# B&R Automation Studio project AAU12Segmenter (part 6)

#### rotationProgram.st
```iecst
ACTION rotationTask:
	positionContainerRotation[0].initXPos := 0.180;
	positionContainerRotation[0].initYPos := 0.060;
	positionContainerRotation[1].initXPos := 0.060;
	positionContainerRotation[1].initYPos := 0.060;
	positionContainerRotation[2].initXPos := 0.060;
	positionContainerRotation[2].initYPos := 0.180;
	positionContainerRotation[3].initXPos := 0.180;
	positionContainerRotation[3].initYPos := 0.180;

	positionContainerRotation[4].initXPos := 0.120;
	positionContainerRotation[4].initYPos := 0.360;
	positionContainerRotation[5].initXPos := 0.360;
	positionContainerRotation[5].initYPos := 0.360;
	positionContainerRotation[6].initXPos := 0.600;
	positionContainerRotation[6].initYPos := 0.360;
	positionContainerRotation[7].initXPos := 0.360;
	positionContainerRotation[7].initYPos := 0.600;

	gWorkStations[0].par.xLocation										:= 0.180;
	gWorkStations[0].par.yLocation										:= 0.060;
	gWorkStations[0].par.nextStationSelector							:= '1';
	gWorkStations[0].par.processTime									:= 0;
	gWorkStations[0].par.pathRouting									:= 1;
	gWorkStations[0].par.landBeforeProcess								:= FALSE;
	gWorkStations[0].par.ArcMovement									:= FALSE;

	gWorkStations[1].par.xLocation										:= 0.060;
	gWorkStations[1].par.yLocation										:= 0.180;
	gWorkStations[1].par.nextStationSelector							:= '0';
	gWorkStations[1].par.processTime									:= 2;
	gWorkStations[1].par.pathRouting									:= 1;
	gWorkStations[1].par.landBeforeProcess								:= TRUE;
	gWorkStations[1].par.ArcMovement									:= FALSE;

	CASE em.substate OF
		14000:
			em.description := 'Move shuttle to pre pos';
			tempShuttleCounter := 0;
			MC_BR_MoveInPlaneAsync_Acp6D_0.Parameters.Acceleration := gAcp6DCtrl.Par.Acceleration;
			MC_BR_MoveInPlaneAsync_Acp6D_0.Parameters.Velocity := gAcp6DCtrl.Par.Velocity;
			FOR i := 0 TO UINT_TO_USINT(localCurrentNumShuttles-1) DO
				MC_BR_MoveInPlaneAsync_Acp6D_0.Parameters.AsyncPar[i].Shuttle := ADR(gAcp6DCtrl.Status.ShuttleInfo[i].shuttleRef);
				MC_BR_MoveInPlaneAsync_Acp6D_0.Parameters.AsyncPar[i].X := positionContainerRotation[i].initXPos;
				MC_BR_MoveInPlaneAsync_Acp6D_0.Parameters.AsyncPar[i].Y := positionContainerRotation[i].initYPos;
			END_FOR
			MC_BR_MoveInPlaneAsync_Acp6D_0.Execute := TRUE;
			IF MC_BR_MoveInPlaneAsync_Acp6D_0.Done THEN
				MC_BR_MoveInPlaneAsync_Acp6D_0.Execute := FALSE;
				tempShuttleCounter := 4;
				em.substate := 14005;
			END_IF

		14005:
			em.description := 'Start rotation of shuttle 5-10';
			IF tempShuttleCounter > localCurrentNumShuttles-1 THEN
				tempShuttleCounter := 0;
				em.substate := 14010;
			ELSE
				MC_BR_RotaryMotionSpin_Acp6D_0.Shuttle := ADR(gAcp6DCtrl.Status.ShuttleInfo[tempShuttleCounter].shuttleRef);
				MC_BR_RotaryMotionSpin_Acp6D_0.Parameters.Acceleration := gAcp6DCtrl.Par.rotationAcceleration;
				MC_BR_RotaryMotionSpin_Acp6D_0.Parameters.Velocity := gAcp6DCtrl.Par.rotationVelocity;
				MC_BR_RotaryMotionSpin_Acp6D_0.Parameters.Duration := 1000;
				MC_BR_RotaryMotionSpin_Acp6D_0.Execute := TRUE;
				IF MC_BR_RotaryMotionSpin_Acp6D_0.Acknowledge THEN
					MC_BR_RotaryMotionSpin_Acp6D_0.Execute := FALSE;
					em.substate := 14006;
				END_IF
			END_IF

		14006:
			em.description := 'Dummy scan';
			TON_0.PT := t#2s;
			TON_0.IN := TRUE;
			IF TON_0.Q THEN
				TON_0.IN := FALSE;
				tempShuttleCounter := tempShuttleCounter + 1;
				em.substate := 14005;
			END_IF

		14010:
			em.description := 'Move shuttle 2 towards workstation 0';
			MC_BR_MoveInPlane_Acp6D_0.Parameters.Acceleration := gAcp6DCtrl.Par.Acceleration;
			MC_BR_MoveInPlane_Acp6D_0.Parameters.Velocity := gAcp6DCtrl.Par.Velocity;
			MC_BR_MoveInPlane_Acp6D_0.Shuttle := ADR(gAcp6DCtrl.Status.ShuttleInfo[1].shuttleRef);;
			MC_BR_MoveInPlane_Acp6D_0.Parameters.Position.X := gWorkStations[0].par.xLocation;;
			MC_BR_MoveInPlane_Acp6D_0.Parameters.Position.Y := gWorkStations[0].par.yLocation;
			MC_BR_MoveInPlane_Acp6D_0.Parameters.Path := 0; //direct
			MC_BR_MoveInPlane_Acp6D_0.Parameters.Mode := 0;
			MC_BR_MoveInPlane_Acp6D_0.Execute := TRUE;
			IF MC_BR_MoveInPlane_Acp6D_0.Acknowledge THEN
				MC_BR_MoveInPlane_Acp6D_0.Execute := FALSE;
				em.substate := 14020;
			END_IF

		14020:
			em.description := 'Move shuttle 3 towards workstation 0';
			MC_BR_MoveInPlane_Acp6D_0.Parameters.Acceleration := gAcp6DCtrl.Par.Acceleration;
			MC_BR_MoveInPlane_Acp6D_0.Parameters.Velocity := gAcp6DCtrl.Par.Velocity;
			MC_BR_MoveInPlane_Acp6D_0.Shuttle := ADR(gAcp6DCtrl.Status.ShuttleInfo[2].shuttleRef);;
			MC_BR_MoveInPlane_Acp6D_0.Parameters.Position.X := gWorkStations[0].par.xLocation;;
			MC_BR_MoveInPlane_Acp6D_0.Parameters.Position.Y := gWorkStations[0].par.yLocation;
			MC_BR_MoveInPlane_Acp6D_0.Parameters.Path := 2; //Y then X
			MC_BR_MoveInPlane_Acp6D_0.Parameters.Mode := 0;
			MC_BR_MoveInPlane_Acp6D_0.Execute := TRUE;
			IF MC_BR_MoveInPlane_Acp6D_0.Acknowledge THEN
				MC_BR_MoveInPlane_Acp6D_0.Execute := FALSE;
				em.substate := 14030;
			END_IF

		14030:
			em.description := 'Move shuttle 4 towards workstation 1';
			MC_BR_MoveInPlane_Acp6D_0.Parameters.Acceleration := gAcp6DCtrl.Par.Acceleration;
			MC_BR_MoveInPlane_Acp6D_0.Parameters.Velocity := gAcp6DCtrl.Par.Velocity;
			MC_BR_MoveInPlane_Acp6D_0.Shuttle := ADR(gAcp6DCtrl.Status.ShuttleInfo[3].shuttleRef);;
			MC_BR_MoveInPlane_Acp6D_0.Parameters.Position.X := 0.060;
			MC_BR_MoveInPlane_Acp6D_0.Parameters.Position.Y := 0.180;
			MC_BR_MoveInPlane_Acp6D_0.Parameters.Path := 0; //direct
			MC_BR_MoveInPlane_Acp6D_0.Parameters.Mode := 0;
			MC_BR_MoveInPlane_Acp6D_0.Execute := TRUE;
			IF MC_BR_MoveInPlane_Acp6D_0.Acknowledge THEN
				MC_BR_MoveInPlane_Acp6D_0.Execute := FALSE;
				em.substate := 14040;
			END_IF

		14040:
			em.description := 'Move shuttle 4 towards workstation 1';
			MC_BR_MoveInPlane_Acp6D_0.Parameters.Acceleration := gAcp6DCtrl.Par.Acceleration;
			MC_BR_MoveInPlane_Acp6D_0.Parameters.Velocity := gAcp6DCtrl.Par.Velocity;
			MC_BR_MoveInPlane_Acp6D_0.Shuttle := ADR(gAcp6DCtrl.Status.ShuttleInfo[3].shuttleRef);;
			MC_BR_MoveInPlane_Acp6D_0.Parameters.Position.X := gWorkStations[0].par.xLocation;
			MC_BR_MoveInPlane_Acp6D_0.Parameters.Position.Y := gWorkStations[0].par.yLocation;
			MC_BR_MoveInPlane_Acp6D_0.Parameters.Path := 2; //direct
			MC_BR_MoveInPlane_Acp6D_0.Parameters.Mode := 0;
			MC_BR_MoveInPlane_Acp6D_0.Execute := TRUE;
			IF MC_BR_MoveInPlane_Acp6D_0.Acknowledge THEN
				MC_BR_MoveInPlane_Acp6D_0.Execute := FALSE;
				em.substate := 14050;
			END_IF

		14050:
			IF em.status.parent.state <> STATE_EXECUTE THEN
				em.substate := 14060;
			END_IF

		14060:
			MC_BR_AsmStop_Acp6D_0.Execute := TRUE;
			IF MC_BR_AsmStop_Acp6D_0.Done THEN
				MC_BR_AsmStop_Acp6D_0.Execute := FALSE;
				em.substate := 14070;
			END_IF

		14070:
			// Wait for shuttles to settle after rotation
			TON_0.PT := t#2s;
			TON_0.IN := TRUE;
			IF TON_0.Q THEN
				TON_0.IN := FALSE;
				tempShuttleCounter := 4;
				em.substate := 14080;
			END_IF

		14080:
			em.description := 'Start rotation of shuttle 5-10';
			IF tempShuttleCounter > localCurrentNumShuttles-1 THEN
				tempShuttleCounter := 0;
				em.substate := 14100;
			ELSIF gAcp6DCtrl.Status.ShuttleInfo[tempShuttleCounter].State = mcACP6D_SH_STATE_IDLING THEN
				MC_BR_RotaryMotion_Acp6D_0.Shuttle := ADR(gAcp6DCtrl.Status.ShuttleInfo[tempShuttleCounter].shuttleRef);
				MC_BR_RotaryMotion_Acp6D_0.Parameters.Acceleration := gAcp6DCtrl.Par.rotationAcceleration;
				MC_BR_RotaryMotion_Acp6D_0.Parameters.Velocity := gAcp6DCtrl.Par.rotationVelocity;
				MC_BR_RotaryMotion_Acp6D_0.Parameters.Mode := mcACP6D_ROTATE_CLOCKWISE;
				MC_BR_RotaryMotion_Acp6D_0.Parameters.Angle := 0;
				MC_BR_RotaryMotion_Acp6D_0.Execute := TRUE;
				IF MC_BR_RotaryMotion_Acp6D_0.Done THEN
					MC_BR_RotaryMotion_Acp6D_0.Execute := FALSE;
					em.substate := 14090;
				END_IF
			END_IF

		14090:
			em.description := 'Dummyscan';
			tempShuttleCounter := tempShuttleCounter + 1;
			em.substate := 14080;

		14100:
			em.description := 'check all shuttles that is rotating to pos zero is done';
			FOR i := 4 TO NUM_SHUTTLES DO
				IF gAcp6DCtrl.Status.ShuttleInfo[i].State = mcACP6D_SH_STATE_IDLING THEN
				ELSE
					EXIT;
				END_IF
			END_FOR
			IF i > NUM_SHUTTLES THEN
				em.substate := 14110;
			END_IF

		14110:
			em.cmd.sc := TRUE;

	END_CASE

END_ACTION

ACTION rotationStation:
	CASE cm.state OF
		// Display station at image
		//'<foreignObject x="20" y="20" width="300" height="300"><img src="Media/statusGreen.png" height="300" width="300"/>'
		//brsstrcat(ADR(showWorkStations),ADR('<foreingObject x="'));
		//brdkStrCat(ADR(showWorkStations), ADR(testDraw));
		//brdkStrCat(ADR(showWorkStations),'<foreingObject x="');

		0:
			//Check what shuttle is on top of workstation
			FOR k := 0 TO NUM_SHUTTLES DO
				IF((gAcp6DCtrl.Status.ShuttleInfo[k].Position.X > pWorkStations.par.xLocation - MARGIN AND gAcp6DCtrl.Status.ShuttleInfo[k].Position.X < pWorkStations.par.xLocation + MARGIN) AND
					gAcp6DCtrl.Status.ShuttleInfo[k].Position.Y > pWorkStations.par.yLocation - MARGIN AND gAcp6DCtrl.Status.ShuttleInfo[k].Position.Y < pWorkStations.par.yLocation + MARGIN) THEN
					IF gAcp6DCtrl.Status.ShuttleInfo[k].State = mcACP6D_SH_STATE_IDLING THEN
						pWorkStations.par.tempShuttleID := k;
						cm.state := 10;
					END_IF
				END_IF
			END_FOR

		10:
			//Move first workstation
			pWorkStations.MC_BR_MoveInPlane_Acp6D_0.Shuttle := ADR(gAcp6DCtrl.Status.ShuttleInfo[pWorkStations.par.tempShuttleID].shuttleRef);
			pWorkStations.MC_BR_MoveInPlane_Acp6D_0.Parameters.Velocity := gAcp6DCtrl.Par.Velocity;
			pWorkStations.MC_BR_MoveInPlane_Acp6D_0.Parameters.Acceleration := gAcp6DCtrl.Par.Acceleration;
			pWorkStations.MC_BR_MoveInPlane_Acp6D_0.Parameters.Position.X := 0.360;
			pWorkStations.MC_BR_MoveInPlane_Acp6D_0.Parameters.Position.Y := 0.120;
			pWorkStations.MC_BR_MoveInPlane_Acp6D_0.Parameters.Mode := 0; //Absolute
			pWorkStations.MC_BR_MoveInPlane_Acp6D_0.Parameters.Path := 1; //0 Diagonal, 1 First X then Y, 2 First Y then X
			pWorkStations.MC_BR_MoveInPlane_Acp6D_0.Execute := TRUE;
			IF pWorkStations.MC_BR_MoveInPlane_Acp6D_0.Done THEN
				pWorkStations.MC_BR_MoveInPlane_Acp6D_0.Execute := FALSE;
				cm.state := 20;
			END_IF

		20:
			//Rotate 90 degress
			em.cmd.sc := FALSE;
			pWorkStations.MC_BR_RotaryMotion_Acp6D_0.Shuttle := ADR(gAcp6DCtrl.Status.ShuttleInfo[pWorkStations.par.tempShuttleID].shuttleRef);
			pWorkStations.MC_BR_RotaryMotion_Acp6D_0.Parameters.Acceleration := gAcp6DCtrl.Par.rotationAcceleration;
			pWorkStations.MC_BR_RotaryMotion_Acp6D_0.Parameters.Velocity := gAcp6DCtrl.Par.rotationVelocity;
			pWorkStations.MC_BR_RotaryMotion_Acp6D_0.Parameters.Angle := 1.57079633; //90 degress
			pWorkStations.MC_BR_RotaryMotion_Acp6D_0.Parameters.Mode := 0;
			pWorkStations.MC_BR_RotaryMotion_Acp6D_0.Execute := TRUE;
			IF pWorkStations.MC_BR_RotaryMotion_Acp6D_0.Done THEN
				pWorkStations.MC_BR_RotaryMotion_Acp6D_0.Execute := FALSE;
				cm.state := 30;
			END_IF

		30:
			//Move
			pWorkStations.MC_BR_MoveInPlane_Acp6D_0.Shuttle := ADR(gAcp6DCtrl.Status.ShuttleInfo[pWorkStations.par.tempShuttleID].shuttleRef);
			pWorkStations.MC_BR_MoveInPlane_Acp6D_0.Parameters.Velocity := gAcp6DCtrl.Par.Velocity;
			pWorkStations.MC_BR_MoveInPlane_Acp6D_0.Parameters.Acceleration := gAcp6DCtrl.Par.Acceleration;
			pWorkStations.MC_BR_MoveInPlane_Acp6D_0.Parameters.Position.X := 0.420;
			pWorkStations.MC_BR_MoveInPlane_Acp6D_0.Parameters.Position.Y := 0.120;
			pWorkStations.MC_BR_MoveInPlane_Acp6D_0.Parameters.Mode := 0; //Absolute
			pWorkStations.MC_BR_MoveInPlane_Acp6D_0.Parameters.Path := 1; //0 Diagonal, 1 First X then Y, 2 First Y then X
			pWorkStations.MC_BR_MoveInPlane_Acp6D_0.Execute := TRUE;
			IF pWorkStations.MC_BR_MoveInPlane_Acp6D_0.Acknowledge THEN
				pWorkStations.MC_BR_MoveInPlane_Acp6D_0.Execute := FALSE;
				cm.state := 40;
			END_IF

		40:
			pWorkStations.TON_0.IN := TRUE;
			pWorkStations.TON_0.PT := t#1s;
			IF pWorkStations.TON_0.Q THEN
				pWorkStations.TON_0.IN := FALSE;
				cm.state := 50;
			END_IF

		50:
			//Move
			pWorkStations.MC_BR_MoveInPlane_Acp6D_0.Shuttle := ADR(gAcp6DCtrl.Status.ShuttleInfo[pWorkStations.par.tempShuttleID].shuttleRef);
			pWorkStations.MC_BR_MoveInPlane_Acp6D_0.Parameters.Velocity := gAcp6DCtrl.Par.Velocity;
			pWorkStations.MC_BR_MoveInPlane_Acp6D_0.Parameters.Acceleration := gAcp6DCtrl.Par.Acceleration;
			pWorkStations.MC_BR_MoveInPlane_Acp6D_0.Parameters.Position.X := 0.360;
			pWorkStations.MC_BR_MoveInPlane_Acp6D_0.Parameters.Position.Y := 0.120;
			pWorkStations.MC_BR_MoveInPlane_Acp6D_0.Parameters.Mode := 0; //Absolute
			pWorkStations.MC_BR_MoveInPlane_Acp6D_0.Parameters.Path := 1; //0 Diagonal, 1 First X then Y, 2 First Y then X
			pWorkStations.MC_BR_MoveInPlane_Acp6D_0.Execute := TRUE;
			IF pWorkStations.MC_BR_MoveInPlane_Acp6D_0.Acknowledge THEN
				pWorkStations.MC_BR_MoveInPlane_Acp6D_0.Execute := FALSE;
				cm.state := 60;
			END_IF

		60:
			//Rotate 90 degress
			em.cmd.sc := FALSE;
			pWorkStations.MC_BR_RotaryMotion_Acp6D_0.Shuttle := ADR(gAcp6DCtrl.Status.ShuttleInfo[pWorkStations.par.tempShuttleID].shuttleRef);
			pWorkStations.MC_BR_RotaryMotion_Acp6D_0.Parameters.Acceleration := gAcp6DCtrl.Par.rotationAcceleration;
			pWorkStations.MC_BR_RotaryMotion_Acp6D_0.Parameters.Velocity := gAcp6DCtrl.Par.rotationVelocity;
			pWorkStations.MC_BR_RotaryMotion_Acp6D_0.Parameters.Angle := 3.14159265; //180 degress
			pWorkStations.MC_BR_RotaryMotion_Acp6D_0.Parameters.Mode := 0;
			pWorkStations.MC_BR_RotaryMotion_Acp6D_0.Execute := TRUE;
			IF pWorkStations.MC_BR_RotaryMotion_Acp6D_0.Done THEN
				pWorkStations.MC_BR_RotaryMotion_Acp6D_0.Execute := FALSE;
				cm.state := 70;
			END_IF

		70:
			//Move
			pWorkStations.MC_BR_MoveInPlane_Acp6D_0.Shuttle := ADR(gAcp6DCtrl.Status.ShuttleInfo[pWorkStations.par.tempShuttleID].shuttleRef);
			pWorkStations.MC_BR_MoveInPlane_Acp6D_0.Parameters.Velocity := gAcp6DCtrl.Par.Velocity;
			pWorkStations.MC_BR_MoveInPlane_Acp6D_0.Parameters.Acceleration := gAcp6DCtrl.Par.Acceleration;
			pWorkStations.MC_BR_MoveInPlane_Acp6D_0.Parameters.Position.X := 0.420;
			pWorkStations.MC_BR_MoveInPlane_Acp6D_0.Parameters.Position.Y := 0.120;
			pWorkStations.MC_BR_MoveInPlane_Acp6D_0.Parameters.Mode := 0; //Absolute
			pWorkStations.MC_BR_MoveInPlane_Acp6D_0.Parameters.Path := 1; //0 Diagonal, 1 First X then Y, 2 First Y then X
			pWorkStations.MC_BR_MoveInPlane_Acp6D_0.Execute := TRUE;
			IF pWorkStations.MC_BR_MoveInPlane_Acp6D_0.Acknowledge THEN
				pWorkStations.MC_BR_MoveInPlane_Acp6D_0.Execute := FALSE;
				cm.state := 80;
			END_IF

		80:
			pWorkStations.TON_0.IN := TRUE;
			pWorkStations.TON_0.PT := t#1s;
			IF pWorkStations.TON_0.Q THEN
				pWorkStations.TON_0.IN := FALSE;
				cm.state := 90;
			END_IF

		90:
			//Move
			pWorkStations.MC_BR_MoveInPlane_Acp6D_0.Shuttle := ADR(gAcp6DCtrl.Status.ShuttleInfo[pWorkStations.par.tempShuttleID].shuttleRef);
			pWorkStations.MC_BR_MoveInPlane_Acp6D_0.Parameters.Velocity := gAcp6DCtrl.Par.Velocity;
			pWorkStations.MC_BR_MoveInPlane_Acp6D_0.Parameters.Acceleration := gAcp6DCtrl.Par.Acceleration;
			pWorkStations.MC_BR_MoveInPlane_Acp6D_0.Parameters.Position.X := 0.360;
			pWorkStations.MC_BR_MoveInPlane_Acp6D_0.Parameters.Position.Y := 0.120;
			pWorkStations.MC_BR_MoveInPlane_Acp6D_0.Parameters.Mode := 0; //Absolute
			pWorkStations.MC_BR_MoveInPlane_Acp6D_0.Parameters.Path := 1; //0 Diagonal, 1 First X then Y, 2 First Y then X
			pWorkStations.MC_BR_MoveInPlane_Acp6D_0.Execute := TRUE;
			IF pWorkStations.MC_BR_MoveInPlane_Acp6D_0.Acknowledge THEN
				pWorkStations.MC_BR_MoveInPlane_Acp6D_0.Execute := FALSE;
				cm.state := 100;
			END_IF

		100:
			//Rotate 90 degress
			em.cmd.sc := FALSE;
			pWorkStations.MC_BR_RotaryMotion_Acp6D_0.Shuttle := ADR(gAcp6DCtrl.Status.ShuttleInfo[pWorkStations.par.tempShuttleID].shuttleRef);
			pWorkStations.MC_BR_RotaryMotion_Acp6D_0.Parameters.Acceleration := gAcp6DCtrl.Par.rotationAcceleration;
			pWorkStations.MC_BR_RotaryMotion_Acp6D_0.Parameters.Velocity := gAcp6DCtrl.Par.rotationVelocity;
			pWorkStations.MC_BR_RotaryMotion_Acp6D_0.Parameters.Angle := 4.71238898; //270 degress
			pWorkStations.MC_BR_RotaryMotion_Acp6D_0.Parameters.Mode := 0;
			pWorkStations.MC_BR_RotaryMotion_Acp6D_0.Execute := TRUE;
			IF pWorkStations.MC_BR_RotaryMotion_Acp6D_0.Done THEN
				pWorkStations.MC_BR_RotaryMotion_Acp6D_0.Execute := FALSE;
				cm.state := 110;
			END_IF

		110:
			//Move
			pWorkStations.MC_BR_MoveInPlane_Acp6D_0.Shuttle := ADR(gAcp6DCtrl.Status.ShuttleInfo[pWorkStations.par.tempShuttleID].shuttleRef);
			pWorkStations.MC_BR_MoveInPlane_Acp6D_0.Parameters.Velocity := gAcp6DCtrl.Par.Velocity;
			pWorkStations.MC_BR_MoveInPlane_Acp6D_0.Parameters.Acceleration := gAcp6DCtrl.Par.Acceleration;
			pWorkStations.MC_BR_MoveInPlane_Acp6D_0.Parameters.Position.X := 0.420;
			pWorkStations.MC_BR_MoveInPlane_Acp6D_0.Parameters.Position.Y := 0.120;
			pWorkStations.MC_BR_MoveInPlane_Acp6D_0.Parameters.Mode := 0; //Absolute
			pWorkStations.MC_BR_MoveInPlane_Acp6D_0.Parameters.Path := 1; //0 Diagonal, 1 First X then Y, 2 First Y then X
			pWorkStations.MC_BR_MoveInPlane_Acp6D_0.Execute := TRUE;
			IF pWorkStations.MC_BR_MoveInPlane_Acp6D_0.Acknowledge THEN
				pWorkStations.MC_BR_MoveInPlane_Acp6D_0.Execute := FALSE;
				cm.state := 120;
			END_IF

		120:
			pWorkStations.TON_0.IN := TRUE;
			pWorkStations.TON_0.PT := t#1s;
			IF pWorkStations.TON_0.Q THEN
				pWorkStations.TON_0.IN := FALSE;
				cm.state := 130;
			END_IF

		130:
			//Move
			pWorkStations.MC_BR_MoveInPlane_Acp6D_0.Shuttle := ADR(gAcp6DCtrl.Status.ShuttleInfo[pWorkStations.par.tempShuttleID].shuttleRef);
			pWorkStations.MC_BR_MoveInPlane_Acp6D_0.Parameters.Velocity := gAcp6DCtrl.Par.Velocity;
			pWorkStations.MC_BR_MoveInPlane_Acp6D_0.Parameters.Acceleration := gAcp6DCtrl.Par.Acceleration;
			pWorkStations.MC_BR_MoveInPlane_Acp6D_0.Parameters.Position.X := 0.360;
			pWorkStations.MC_BR_MoveInPlane_Acp6D_0.Parameters.Position.Y := 0.120;
			pWorkStations.MC_BR_MoveInPlane_Acp6D_0.Parameters.Mode := 0; //Absolute
			pWorkStations.MC_BR_MoveInPlane_Acp6D_0.Parameters.Path := 1; //0 Diagonal, 1 First X then Y, 2 First Y then X
			pWorkStations.MC_BR_MoveInPlane_Acp6D_0.Execute := TRUE;
			IF pWorkStations.MC_BR_MoveInPlane_Acp6D_0.Acknowledge THEN
				pWorkStations.MC_BR_MoveInPlane_Acp6D_0.Execute := FALSE;
				cm.state := 140;
			END_IF

		140:
			//Rotate
			em.cmd.sc := FALSE;
			pWorkStations.MC_BR_RotaryMotion_Acp6D_0.Shuttle := ADR(gAcp6DCtrl.Status.ShuttleInfo[pWorkStations.par.tempShuttleID].shuttleRef);
			pWorkStations.MC_BR_RotaryMotion_Acp6D_0.Parameters.Acceleration := gAcp6DCtrl.Par.rotationAcceleration;
			pWorkStations.MC_BR_RotaryMotion_Acp6D_0.Parameters.Velocity := gAcp6DCtrl.Par.rotationVelocity; //RPM
			pWorkStations.MC_BR_RotaryMotion_Acp6D_0.Parameters.Angle := 0; //0 degress
			pWorkStations.MC_BR_RotaryMotion_Acp6D_0.Parameters.Mode := 1;
			pWorkStations.MC_BR_RotaryMotion_Acp6D_0.Execute := TRUE;
			IF pWorkStations.MC_BR_RotaryMotion_Acp6D_0.Done THEN
				pWorkStations.MC_BR_RotaryMotion_Acp6D_0.Execute := FALSE;
				cm.state := 150;
			END_IF

//		145:
//			em.cmd.sc := FALSE;
//			pWorkStations.MC_BR_RotaryMotionSpin_Acp6D_0.Shuttle := ADR(gAcp6DCtrl.Status.ShuttleInfo[pWorkStations.par.tempShuttleID].shuttleRef);
//			pWorkStations.MC_BR_RotaryMotionSpin_Acp6D_0.Parameters.Acceleration := gAcp6DCtrl.Par.Acceleration;
//			pWorkStations.MC_BR_RotaryMotionSpin_Acp6D_0.Parameters.Velocity := 200; //RPM
//			pWorkStations.MC_BR_RotaryMotionSpin_Acp6D_0.Parameters.Duration := 5;
//			pWorkStations.MC_BR_RotaryMotionSpin_Acp6D_0.Execute := TRUE;
//			IF pWorkStations.MC_BR_RotaryMotionSpin_Acp6D_0.Done THEN
//				pWorkStations.MC_BR_RotaryMotionSpin_Acp6D_0.Execute := FALSE;
//				cm.state := 150;
//			END_IF

		150:
			//Move
			pWorkStations.MC_BR_MoveInPlane_Acp6D_0.Shuttle := ADR(gAcp6DCtrl.Status.ShuttleInfo[pWorkStations.par.tempShuttleID].shuttleRef);
			pWorkStations.MC_BR_MoveInPlane_Acp6D_0.Parameters.Velocity := gAcp6DCtrl.Par.Velocity;
			pWorkStations.MC_BR_MoveInPlane_Acp6D_0.Parameters.Acceleration := gAcp6DCtrl.Par.Acceleration;
			pWorkStations.MC_BR_MoveInPlane_Acp6D_0.Parameters.Position.X := 0.060;
			pWorkStations.MC_BR_MoveInPlane_Acp6D_0.Parameters.Position.Y := 0.180;
			pWorkStations.MC_BR_MoveInPlane_Acp6D_0.Parameters.Mode := 0; //Absolute
			pWorkStations.MC_BR_MoveInPlane_Acp6D_0.Parameters.Path := 2; //0 Diagonal, 1 First X then Y, 2 First Y then X
			pWorkStations.MC_BR_MoveInPlane_Acp6D_0.Execute := TRUE;
			IF pWorkStations.MC_BR_MoveInPlane_Acp6D_0.Acknowledge THEN
				pWorkStations.MC_BR_MoveInPlane_Acp6D_0.Execute := FALSE;
				cm.state := 160;
			END_IF

		160:
			//Move
			pWorkStations.MC_BR_MoveInPlane_Acp6D_0.Shuttle := ADR(gAcp6DCtrl.Status.ShuttleInfo[pWorkStations.par.tempShuttleID].shuttleRef);
			pWorkStations.MC_BR_MoveInPlane_Acp6D_0.Parameters.Velocity := gAcp6DCtrl.Par.Velocity;
			pWorkStations.MC_BR_MoveInPlane_Acp6D_0.Parameters.Acceleration := gAcp6DCtrl.Par.Acceleration;
			pWorkStations.MC_BR_MoveInPlane_Acp6D_0.Parameters.Position.X := gWorkStations[0].par.xLocation;
			pWorkStations.MC_BR_MoveInPlane_Acp6D_0.Parameters.Position.Y := gWorkStations[0].par.yLocation;
			pWorkStations.MC_BR_MoveInPlane_Acp6D_0.Parameters.Mode := 0; //Absolute
			pWorkStations.MC_BR_MoveInPlane_Acp6D_0.Parameters.Path := 2; //0 Diagonal, 1 First X then Y, 2 First Y then X
			pWorkStations.MC_BR_MoveInPlane_Acp6D_0.Execute := TRUE;
			IF pWorkStations.MC_BR_MoveInPlane_Acp6D_0.Acknowledge THEN
				pWorkStations.MC_BR_MoveInPlane_Acp6D_0.Execute := FALSE;
				cm.state := 0;
			END_IF

	END_CASE

	//Calls
	pWorkStations.MC_BR_MoveInPlane_Acp6D_0();
	pWorkStations.MC_BR_MoveArc_Acp6D_0();
	pWorkStations.MC_BR_ShLevitation_Acp6D_0();
	pWorkStations.MC_BR_RotaryMotion_Acp6D_0();
	pWorkStations.MC_BR_RotaryMotionSpin_Acp6D_0();
	pWorkStations.TON_0();
	cm();

END_ACTION
```

#### steelSheet.st
```iecst
ACTION steelSheetTask:
	positionContainerSteelSheet[0].initXPos := 0.300;
	positionContainerSteelSheet[0].initYPos := 0.060;
	positionContainerSteelSheet[1].initXPos := 0.420;
	positionContainerSteelSheet[1].initYPos := 0.060;
	positionContainerSteelSheet[2].initXPos := 0.540;
	positionContainerSteelSheet[2].initYPos := 0.060;
	positionContainerSteelSheet[3].initXPos := 0.660;
	positionContainerSteelSheet[3].initYPos := 0.060;

	positionContainerSteelSheet[4].initXPos := 0.540;
	positionContainerSteelSheet[4].initYPos := 0.900;
	positionContainerSteelSheet[5].initXPos := 0.660;
	positionContainerSteelSheet[5].initYPos := 0.900;
	positionContainerSteelSheet[6].initXPos := 0.540;
	positionContainerSteelSheet[6].initYPos := 0.780;
	positionContainerSteelSheet[7].initXPos := 0.660;
	positionContainerSteelSheet[7].initYPos := 0.780;

	gWorkstations[0].par.xLocation										:= 0.300;
	gWorkstations[0].par.yLocation										:= 0.060;
	gWorkstations[0].par.nextStationSelector							:= '0';
	gWorkstations[0].par.processTime									:= 0;
	gWorkstations[0].par.pathRouting									:= 0;
	gWorkstations[0].par.landBeforeProcess								:= FALSE;
	gWorkstations[0].par.ArcMovement									:= FALSE;

	gWorkstations[1].par.xLocation										:= 0.420;
	gWorkstations[1].par.yLocation										:= 0.060;
	gWorkstations[1].par.nextStationSelector							:= '1';
	gWorkstations[1].par.processTime									:= 0;
	gWorkstations[1].par.pathRouting									:= 0;
	gWorkstations[1].par.landBeforeProcess								:= FALSE;
	gWorkstations[1].par.ArcMovement									:= FALSE;

	gWorkstations[2].par.xLocation										:= 0.540;
	gWorkstations[2].par.yLocation										:= 0.060;
	gWorkstations[2].par.nextStationSelector							:= '2';
	gWorkstations[2].par.processTime									:= 0;
	gWorkstations[2].par.pathRouting									:= 0;
	gWorkstations[2].par.landBeforeProcess								:= FALSE;
	gWorkstations[2].par.ArcMovement									:= FALSE;

	gWorkstations[3].par.xLocation										:= 0.660;
	gWorkstations[3].par.yLocation										:= 0.060;
	gWorkstations[3].par.nextStationSelector							:= '3';
	gWorkstations[3].par.processTime									:= 0;
	gWorkstations[3].par.pathRouting									:= 0;
	gWorkstations[3].par.landBeforeProcess								:= FALSE;
	gWorkstations[3].par.ArcMovement									:= FALSE;

	CASE em.substate OF
		15000:
			em.description := 'Move shuttle to pre pos';
			tempShuttleCounter := 0;
			MC_BR_MoveInPlaneAsync_Acp6D_0.Parameters.Acceleration := gAcp6DCtrl.Par.Acceleration;
			MC_BR_MoveInPlaneAsync_Acp6D_0.Parameters.Velocity := gAcp6DCtrl.Par.Velocity;
			FOR i := 0 TO UINT_TO_USINT(localCurrentNumShuttles-1) DO
				MC_BR_MoveInPlaneAsync_Acp6D_0.Parameters.AsyncPar[i].Shuttle := ADR(gAcp6DCtrl.Status.ShuttleInfo[i].shuttleRef);
				MC_BR_MoveInPlaneAsync_Acp6D_0.Parameters.AsyncPar[i].X := positionContainerSteelSheet[i].initXPos;
				MC_BR_MoveInPlaneAsync_Acp6D_0.Parameters.AsyncPar[i].Y := positionContainerSteelSheet[i].initYPos;
			END_FOR
			MC_BR_MoveInPlaneAsync_Acp6D_0.Execute := TRUE;
			IF MC_BR_MoveInPlaneAsync_Acp6D_0.Acknowledge THEN
				MC_BR_MoveInPlaneAsync_Acp6D_0.Execute := FALSE;
				em.substate := 15010;
			END_IF

		15010:
			em.description := 'Shuttle moves at a higher levitation hight';

	END_CASE

END_ACTION

ACTION steelSheetStation:
	CASE cm.state OF
		0:
			//Check what shuttle is on top of workstation
			FOR k := 0 TO NUM_SHUTTLES DO
				IF((gAcp6DCtrl.Status.ShuttleInfo[k].Position.X > pWorkstation.par.xLocation - MARGIN AND gAcp6DCtrl.Status.ShuttleInfo[k].Position.X < pWorkstation.par.xLocation + MARGIN) AND
					gAcp6DCtrl.Status.ShuttleInfo[k].Position.Y > pWorkstation.par.yLocation - MARGIN AND gAcp6DCtrl.Status.ShuttleInfo[k].Position.Y < pWorkstation.par.yLocation + MARGIN) THEN
					IF gAcp6DCtrl.Status.ShuttleInfo[k].State = mcACP6D_SH_STATE_IDLING THEN
						pWorkstation.par.tempShuttleID := k;
						cm.state := 10;
					END_IF
				END_IF
			END_FOR

		10:
			pWorkstation.MC_BR_Move6D_Acp6D_0.Shuttle := ADR(gAcp6DCtrl.Status.ShuttleInfo[pWorkstation.par.tempShuttleID].shuttleRef);
			pWorkstation.MC_BR_Move6D_Acp6D_0.Parameters.InPlane.Velocity := 0.1;
			pWorkstation.MC_BR_Move6D_Acp6D_0.Parameters.InPlane.Acceleration := 0.1;
			pWorkstation.MC_BR_Move6D_Acp6D_0.Parameters.InPlane.Position.X := pWorkstation.par.xLocation;
			pWorkstation.MC_BR_Move6D_Acp6D_0.Parameters.InPlane.Position.Y := 0.180;
			pWorkstation.MC_BR_Move6D_Acp6D_0.Parameters.ShortAxis.Position.Z := steelSheetFlyingHeight;
			pWorkstation.MC_BR_Move6D_Acp6D_0.Parameters.ShortAxis.Position.Rx := 0;
			pWorkstation.MC_BR_Move6D_Acp6D_0.Parameters.ShortAxis.Position.Ry := 0;
			pWorkstation.MC_BR_Move6D_Acp6D_0.Parameters.ShortAxis.Position.Rz := 0;
			pWorkstation.MC_BR_Move6D_Acp6D_0.Execute := TRUE;
			IF pWorkstation.MC_BR_Move6D_Acp6D_0.Done THEN
				pWorkstation.MC_BR_Move6D_Acp6D_0.Execute := FALSE;
				cm.state := 30;
			END_IF

		30:
			pWorkstation.MC_BR_Move6D_Acp6D_0.Shuttle := ADR(gAcp6DCtrl.Status.ShuttleInfo[pWorkstation.par.tempShuttleID].shuttleRef);
			pWorkstation.MC_BR_Move6D_Acp6D_0.Parameters.InPlane.Velocity := 0.1;
			pWorkstation.MC_BR_Move6D_Acp6D_0.Parameters.InPlane.Acceleration := 0.1;
			pWorkstation.MC_BR_Move6D_Acp6D_0.Parameters.InPlane.Position.X := pWorkstation.par.xLocation;
			pWorkstation.MC_BR_Move6D_Acp6D_0.Parameters.InPlane.Position.Y := 0.060;
			pWorkstation.MC_BR_Move6D_Acp6D_0.Parameters.ShortAxis.Position.Rx := 0;
			pWorkstation.MC_BR_Move6D_Acp6D_0.Parameters.ShortAxis.Position.Ry := 0;
			pWorkstation.MC_BR_Move6D_Acp6D_0.Parameters.ShortAxis.Position.Rz := 0;
			pWorkstation.MC_BR_Move6D_Acp6D_0.Parameters.ShortAxis.Position.Z := steelSheetFlyingHeight;
			pWorkstation.MC_BR_Move6D_Acp6D_0.Execute := TRUE;
			IF pWorkstation.MC_BR_Move6D_Acp6D_0.Done THEN
				pWorkstation.MC_BR_Move6D_Acp6D_0.Execute := FALSE;
				cm.state := 0;
			END_IF

	END_CASE

	//Calls
	pWorkstation.MC_BR_MoveInPlane_Acp6D_0();
	pWorkstation.MC_BR_MoveArc_Acp6D_0();
	pWorkstation.MC_BR_Move6D_Acp6D_0();
	pWorkstation.MC_BR_ShLevitation_Acp6D_0();
	pWorkstation.MC_BR_RotaryMotion_Acp6D_0();
	pWorkstation.MC_BR_RotaryMotionSpin_Acp6D_0();
	pWorkstation.TON_0();
	cm();

END_ACTION
```

#### Test.st
```iecst
ACTION testProgram:
//setup
	positionContainerTestProgram[0].initXPos := 0.050;
	positionContainerTestProgram[0].initYPos := 0.060;

	positionContainerTestProgram[1].initXPos := 0.050;
	positionContainerTestProgram[1].initYPos := 0.180;

	positionContainerTestProgram[2].initXPos := 0.050;
	positionContainerTestProgram[2].initYPos := 0.300;

	positionContainerTestProgram[3].initXPos := 0.050;
	positionContainerTestProgram[3].initYPos := 0.420;

	positionContainerTestProgram[4].initXPos := 0.660;
	positionContainerTestProgram[4].initYPos := 0.900;

	positionContainerTestProgram[5].initXPos := 0.660;
	positionContainerTestProgram[5].initYPos := 0.780;

	positionContainerTestProgram[6].initXPos := 0.540;
	positionContainerTestProgram[6].initYPos := 0.900;

	positionContainerTestProgram[7].initXPos := 0.540;
	positionContainerTestProgram[7].initYPos := 0.780;

	CASE em.substate OF
		16000:
			em.description := 'Move shuttles to pre pos';
			MC_BR_MoveInPlaneAsync_Acp6D_0.Parameters.Acceleration := gAcp6DCtrl.Par.Acceleration;
			MC_BR_MoveInPlaneAsync_Acp6D_0.Parameters.Velocity := gAcp6DCtrl.Par.Velocity;
			FOR i := 0 TO NUM_SHUTTLES DO
				MC_BR_MoveInPlaneAsync_Acp6D_0.Parameters.AsyncPar[i].Shuttle := ADR(gAcp6DCtrl.Status.ShuttleInfo[i].shuttleRef);
				MC_BR_MoveInPlaneAsync_Acp6D_0.Parameters.AsyncPar[i].X := positionContainerTestProgram[i].initXPos;
				MC_BR_MoveInPlaneAsync_Acp6D_0.Parameters.AsyncPar[i].Y := positionContainerTestProgram[i].initYPos;
			END_FOR
			MC_BR_MoveInPlaneAsync_Acp6D_0.Execute := TRUE;
			IF MC_BR_MoveInPlaneAsync_Acp6D_0.Done THEN
				MC_BR_MoveInPlaneAsync_Acp6D_0.Execute := FALSE;
				em.substate := 16010;
			END_IF

		16010:
			em.description := 'Move shuttles in a staircase movement';

	END_CASE

END_ACTION

ACTION testMovements:

	CASE cm.state OF
		0:
			cm.description := 'Start linear movement of the four shuttles';
			pShuttle.function.MC_BR_MoveInPlane_Acp6D_0.Shuttle := ADR(gAcp6DCtrl.Status.ShuttleInfo[pShuttle.par.shuttleID].shuttleRef);

			pShuttle.function.MC_BR_MoveInPlane_Acp6D_0.Parameters.Mode         := 0; //Absolute movement
			pShuttle.function.MC_BR_MoveInPlane_Acp6D_0.Parameters.Position.X   := positionContainerTestProgram[pShuttle.par.shuttleID].initXPos + (USINT_TO_REAL(pShuttle.par.shuttleID)+1)*0.120;
			pShuttle.function.MC_BR_MoveInPlane_Acp6D_0.Parameters.Position.Y   := positionContainerTestProgram[pShuttle.par.shuttleID].initYPos - (USINT_TO_REAL(pShuttle.par.shuttleID))*0.120;
			pShuttle.function.MC_BR_MoveInPlane_Acp6D_0.Parameters.Acceleration := 1.0;
			pShuttle.function.MC_BR_MoveInPlane_Acp6D_0.Parameters.Velocity     := 0.8;
			pShuttle.function.MC_BR_MoveInPlane_Acp6D_0.Parameters.EndVelocity  := 0.0;
			pShuttle.function.MC_BR_MoveInPlane_Acp6D_0.Parameters.Path         := 1; //mcACP6D_PATH_X_THEN_Y

			pShuttle.function.MC_BR_MoveInPlane_Acp6D_0.Execute := TRUE;
			IF pShuttle.function.MC_BR_MoveInPlane_Acp6D_0.Done THEN  // Try to change to DONE
				pShuttle.function.MC_BR_MoveInPlane_Acp6D_0.Execute := FALSE;
				cm.state := 10;
			END_IF

		10:
			cm.description := 'Check if position is reached';
			testObj.targetReached[pShuttle.par.shuttleID] := TRUE;
			cm.state := 15;

		15:
			cm.description := 'Waiting to move back to start position';
			IF testObj.targetReached[0] AND testObj.targetReached[1] AND testObj.targetReached[2] AND testObj.targetReached[3] THEN
				//IF testObj.targetReached[i] THEN
				cm.state := 16;
			END_IF

		16:
			cm.description := 'Setting all targetReached to false';
			testObj.targetReached[pShuttle.par.shuttleID] := FALSE;
			cm.state := 20;

		20:
			cm.description := 'Moving back to the starting position';
			pShuttle.function.MC_BR_MoveInPlane_Acp6D_0.Shuttle := ADR(gAcp6DCtrl.Status.ShuttleInfo[pShuttle.par.shuttleID].shuttleRef);

			pShuttle.function.MC_BR_MoveInPlane_Acp6D_0.Parameters.Mode         := 1; //Relative movement
			pShuttle.function.MC_BR_MoveInPlane_Acp6D_0.Parameters.Position.X   := -(USINT_TO_REAL(pShuttle.par.shuttleID)+1)*0.120;
			pShuttle.function.MC_BR_MoveInPlane_Acp6D_0.Parameters.Position.Y   := (USINT_TO_REAL(pShuttle.par.shuttleID))*0.120;
			pShuttle.function.MC_BR_MoveInPlane_Acp6D_0.Parameters.Acceleration := 1.0;
			pShuttle.function.MC_BR_MoveInPlane_Acp6D_0.Parameters.Velocity     := 0.8;
			pShuttle.function.MC_BR_MoveInPlane_Acp6D_0.Parameters.EndVelocity  := 0.0;
			pShuttle.function.MC_BR_MoveInPlane_Acp6D_0.Parameters.Path         := 2; //mcACP6D_PATH_Y_THEN_X

			pShuttle.function.MC_BR_MoveInPlane_Acp6D_0.Execute := TRUE;
			IF pShuttle.function.MC_BR_MoveInPlane_Acp6D_0.Acknowledge THEN  // Try to change to DONE
				pShuttle.function.MC_BR_MoveInPlane_Acp6D_0.Execute := FALSE;
				cm.state := 30;
			END_IF

		30:
			cm.description := 'Check if position is reached';
			IF gAcp6DCtrl.Status.ShuttleInfo[pShuttle.par.shuttleID].Position.X < positionContainerTestProgram[pShuttle.par.shuttleID].initXPos + 0.001 AND
				gAcp6DCtrl.Status.ShuttleInfo[pShuttle.par.shuttleID].Position.Y > positionContainerTestProgram[pShuttle.par.shuttleID].initYPos - 0.001 THEN
				testObj.targetReached[pShuttle.par.shuttleID] := TRUE;
				cm.state := 35;
			END_IF

		35:
			cm.description := 'Waiting to go back to start of loop';
			IF testObj.targetReached[0] AND testObj.targetReached[1] AND testObj.targetReached[2] AND testObj.targetReached[3] THEN
				//IF testObj.targetReached[i] THEN
				cm.state := 36;
			END_IF

		36:
			cm.description := 'Setting all targetReached to false';
			testObj.targetReached[pShuttle.par.shuttleID] := FALSE;
			cm.state := 0;

	END_CASE

	cm();
	pShuttle.function.MC_BR_MoveInPlane_Acp6D_0();

END_ACTION
```

#### SmartLabSetup.st
```iecst
ACTION smartLabWorkstationSetup:
	// Reset all workstations
	FOR i := 0 TO NR_OF_WORKSTATIONS DO
		gWorkstations[i].par.xLocation				:= 0.0;
		gWorkstations[i].par.yLocation				:= 0.0;
		gWorkstations[i].par.approachPosX			:= 0.0;
		gWorkstations[i].par.approachPosY			:= 0.0;
		gWorkstations[i].par.departPosX				:= 0.0;
		gWorkstations[i].par.departPosY				:= 0.0;
		gWorkstations[i].par.nextStationSelector	:= '0';
		gWorkstations[i].par.processTime			:= 0;
		gWorkstations[i].par.pathRouting			:= 0;
		gWorkstations[i].par.ArcMovement			:= FALSE;
		gWorkstations[i].par.landBeforeProcess		:= FALSE;
	END_FOR

	gWorkstations[0].par.xLocation					:= QuadrantIdxToPos(5);
	gWorkstations[0].par.yLocation					:= QuadrantIdxToPos(0);
	gWorkstations[0].par.approachPosX				:= QuadrantIdxToPos(4);
	gWorkstations[0].par.approachPosY				:= QuadrantIdxToPos(0);
	gWorkstations[0].par.departPosX					:= QuadrantIdxToPos(4);
	gWorkstations[0].par.departPosY					:= QuadrantIdxToPos(1);
	gWorkstations[0].par.nextStationSelector		:= '1';
	gWorkstations[0].par.processTime				:= 1.0;
	gWorkstations[0].par.pathRouting				:= 2;
	gWorkstations[0].par.ArcMovement				:= FALSE;
	gWorkstations[0].par.landBeforeProcess			:= FALSE;

	gWorkstations[1].par.xLocation					:= QuadrantIdxToPos(5);
	gWorkstations[1].par.yLocation					:= QuadrantIdxToPos(3);
	gWorkstations[1].par.approachPosX				:= QuadrantIdxToPos(4);
	gWorkstations[1].par.approachPosY				:= QuadrantIdxToPos(2);
	gWorkstations[1].par.departPosX					:= QuadrantIdxToPos(4);
	gWorkstations[1].par.departPosY					:= QuadrantIdxToPos(4);
	gWorkstations[1].par.nextStationSelector		:= '2';
	gWorkstations[1].par.processTime				:= 1.0;
	gWorkstations[1].par.pathRouting				:= 2;
	gWorkstations[1].par.ArcMovement				:= FALSE;
	gWorkstations[1].par.landBeforeProcess			:= FALSE;

	gWorkstations[2].par.xLocation					:= QuadrantIdxToPos(5);
	gWorkstations[2].par.yLocation					:= QuadrantIdxToPos(6);
	gWorkstations[2].par.approachPosX				:= QuadrantIdxToPos(4);
	gWorkstations[2].par.approachPosY				:= QuadrantIdxToPos(5);
	gWorkstations[2].par.departPosX					:= QuadrantIdxToPos(4);
	gWorkstations[2].par.departPosY					:= QuadrantIdxToPos(7);
	gWorkstations[2].par.nextStationSelector		:= '3';
	gWorkstations[2].par.processTime				:= 1.0;
	gWorkstations[2].par.pathRouting				:= 1;
	gWorkstations[2].par.ArcMovement				:= FALSE;
	gWorkstations[2].par.landBeforeProcess			:= FALSE;

	gWorkstations[3].par.xLocation					:= QuadrantIdxToPos(0);
	gWorkstations[3].par.yLocation					:= QuadrantIdxToPos(6);
	gWorkstations[3].par.approachPosX				:= QuadrantIdxToPos(1);
	gWorkstations[3].par.approachPosY				:= QuadrantIdxToPos(7);
	gWorkstations[3].par.departPosX					:= QuadrantIdxToPos(1);
	gWorkstations[3].par.departPosY					:= QuadrantIdxToPos(5);
	gWorkstations[3].par.nextStationSelector		:= '4';
	gWorkstations[3].par.processTime				:= 1.0;
	gWorkstations[3].par.pathRouting				:= 2;
	gWorkstations[3].par.ArcMovement				:= FALSE;
	gWorkstations[3].par.landBeforeProcess			:= FALSE;

	gWorkstations[4].par.xLocation					:= QuadrantIdxToPos(0);
	gWorkstations[4].par.yLocation					:= QuadrantIdxToPos(3);
	gWorkstations[4].par.approachPosX				:= QuadrantIdxToPos(1);
	gWorkstations[4].par.approachPosY				:= QuadrantIdxToPos(4);
	gWorkstations[4].par.departPosX					:= QuadrantIdxToPos(1);
	gWorkstations[4].par.departPosY					:= QuadrantIdxToPos(2);
	gWorkstations[4].par.nextStationSelector		:= '5';
	gWorkstations[4].par.processTime				:= 1.0;
	gWorkstations[4].par.pathRouting				:= 2;
	gWorkstations[4].par.ArcMovement				:= FALSE;
	gWorkstations[4].par.landBeforeProcess			:= FALSE;

	gWorkstations[5].par.xLocation					:= QuadrantIdxToPos(0);
	gWorkstations[5].par.yLocation					:= QuadrantIdxToPos(0);
	gWorkstations[5].par.approachPosX				:= QuadrantIdxToPos(1);
	gWorkstations[5].par.approachPosY				:= QuadrantIdxToPos(1);
	gWorkstations[5].par.departPosX					:= QuadrantIdxToPos(1);
	gWorkstations[5].par.departPosY					:= QuadrantIdxToPos(0);
	gWorkstations[5].par.nextStationSelector		:= '0';
	gWorkstations[5].par.processTime				:= 1.0;
	gWorkstations[5].par.pathRouting				:= 1;
	gWorkstations[5].par.ArcMovement				:= FALSE;
	gWorkstations[5].par.landBeforeProcess			:= FALSE;

END_ACTION

ACTION smartLabSetup:

	positionContainerSmartLabProgram[0].initXPos := gWorkstations[0].par.xLocation;
	positionContainerSmartLabProgram[0].initYPos := gWorkstations[0].par.yLocation;

	positionContainerSmartLabProgram[1].initXPos := gWorkstations[0].par.xLocation - 1*0.120;
	positionContainerSmartLabProgram[1].initYPos := gWorkstations[0].par.yLocation;

	positionContainerSmartLabProgram[2].initXPos := gWorkstations[0].par.xLocation - 2*0.120;
	positionContainerSmartLabProgram[2].initYPos := gWorkstations[0].par.yLocation;

	positionContainerSmartLabProgram[3].initXPos := gWorkstations[1].par.xLocation;
	positionContainerSmartLabProgram[3].initYPos := gWorkstations[1].par.yLocation;

	positionContainerSmartLabProgram[4].initXPos := gWorkstations[2].par.xLocation;
	positionContainerSmartLabProgram[4].initYPos := gWorkstations[2].par.yLocation;

	positionContainerSmartLabProgram[5].initXPos := gWorkstations[3].par.xLocation;
	positionContainerSmartLabProgram[5].initYPos := gWorkstations[3].par.yLocation;

	positionContainerSmartLabProgram[6].initXPos := gWorkstations[4].par.xLocation;
	positionContainerSmartLabProgram[6].initYPos := gWorkstations[4].par.yLocation;

	positionContainerSmartLabProgram[7].initXPos := gWorkstations[5].par.xLocation;
	positionContainerSmartLabProgram[7].initYPos := gWorkstations[5].par.yLocation;

	smartLabWorkstationSetup; // Setup workstations

	CASE em.substate OF
		17000:
			em.description := 'Resetting parameters';
			FOR i := 0 TO NUM_SHUTTLES DO
				gShuttles[i].cm.state := 0;
				gWorkstations[i].cm.state := 0;

				gWorkstations[i].par.tempShuttleID := -1;
				gShuttles[i].par.tempHighwayColumn := -1;
				shuttlePlans[i].isActive := FALSE;
			END_FOR

			FOR i := 0 TO 3 DO // Highway columns
				FOR k := 0 TO 7 DO // Highway rows
					occupiedPosition[i, k] := FALSE;
				END_FOR
			END_FOR

			TON_0.IN := FALSE;
			bufferSize := SIZEOF(orderBuffer)/SIZEOF(orderBuffer[0]);
			activeShuttles := 0;
			tempShuttleIndex := 1;
			em.substate := 17005;

		17005:
			em.description := 'Move shuttles to pre pos';
			MC_BR_MoveInPlaneAsync_Acp6D_0.Parameters.Acceleration := gAcp6DCtrl.Par.Acceleration;
			MC_BR_MoveInPlaneAsync_Acp6D_0.Parameters.Velocity := gAcp6DCtrl.Par.Velocity;
			FOR i := 0 TO UINT_TO_USINT(localCurrentNumShuttles-1) DO
				MC_BR_MoveInPlaneAsync_Acp6D_0.Parameters.AsyncPar[i].Shuttle := ADR(gAcp6DCtrl.Status.ShuttleInfo[i].shuttleRef);
				MC_BR_MoveInPlaneAsync_Acp6D_0.Parameters.AsyncPar[i].X := positionContainerSmartLabProgram[i].initXPos;
				MC_BR_MoveInPlaneAsync_Acp6D_0.Parameters.AsyncPar[i].Y := positionContainerSmartLabProgram[i].initYPos;
			END_FOR
			MC_BR_MoveInPlaneAsync_Acp6D_0.Execute := TRUE;
			IF MC_BR_MoveInPlaneAsync_Acp6D_0.Done THEN
				MC_BR_MoveInPlaneAsync_Acp6D_0.Execute := FALSE;
				em.substate := 17008;
			END_IF

		17008:
			em.description := 'Move shuttle 2 and 3 towards workstation 0';
			gShuttles[tempShuttleIndex].function.MC_BR_MoveInPlane_Acp6D_0.Shuttle := ADR(gAcp6DCtrl.Status.ShuttleInfo[tempShuttleIndex].shuttleRef);
			gShuttles[tempShuttleIndex].function.MC_BR_MoveInPlane_Acp6D_0.Parameters.Velocity := gAcp6DCtrl.Par.Velocity;
			gShuttles[tempShuttleIndex].function.MC_BR_MoveInPlane_Acp6D_0.Parameters.Acceleration := gAcp6DCtrl.Par.Acceleration;
			gShuttles[tempShuttleIndex].function.MC_BR_MoveInPlane_Acp6D_0.Parameters.Mode := 0; // Absolute
			gShuttles[tempShuttleIndex].function.MC_BR_MoveInPlane_Acp6D_0.Parameters.Path := 1; // X THEN Y

			gShuttles[tempShuttleIndex].function.MC_BR_MoveInPlane_Acp6D_0.Parameters.Position.X := gWorkstations[0].par.xLocation;
			gShuttles[tempShuttleIndex].function.MC_BR_MoveInPlane_Acp6D_0.Parameters.Position.Y := gWorkstations[0].par.yLocation;
			gShuttles[tempShuttleIndex].function.MC_BR_MoveInPlane_Acp6D_0.Execute := TRUE;
			IF gShuttles[tempShuttleIndex].function.MC_BR_MoveInPlane_Acp6D_0.Acknowledge THEN
				gShuttles[tempShuttleIndex].function.MC_BR_MoveInPlane_Acp6D_0.Execute := FALSE;

				IF tempShuttleIndex = 2 THEN
					em.substate := 17010;
				END_IF

				tempShuttleIndex := tempShuttleIndex + 1;
			END_IF

			gShuttles[tempShuttleIndex].function.MC_BR_MoveInPlane_Acp6D_0();

	END_CASE

END_ACTION
```

#### SmartLabBuffer.st
```iecst
ACTION writeOrder:

	orderBuffer[writeIndex] := tempProductOrder;
	//orderBuffer[writeIndex].ID := orderBuffer[writeIndex].ID + 1; // Seems wrong - shouldn't it be orderBuffer[writeIndex].ID := orderBuffer[writeIndex-1].ID + 1?
	bufferEmpty := FALSE;
	writeIndex := (writeIndex + 1) MOD bufferSize;

	IF (writeIndex MOD bufferSize) = readIndex THEN

		bufferFull := TRUE;

	ELSE

		bufferFull := FALSE;

	END_IF

END_ACTION

ACTION readOrder:

	IF NOT bufferEmpty THEN

		productOrder := orderBuffer[readIndex];
		readIndex := (readIndex + 1) MOD bufferSize;
		bufferFull := FALSE;

	END_IF

	// Check if the buffer is empty
	IF (readIndex = writeIndex) AND NOT bufferFull THEN

		bufferEmpty := TRUE;

	ELSE

		bufferEmpty := FALSE;

	END_IF

	//
//	IF (NOT readIndex = writeIndex) OR bufferFull THEN
//
//		productOrder := orderBuffer[readIndex];
//		readIndex := (readIndex + 1) MOD bufferSize;
//		bufferFull := FALSE;
//
//	END_IF

END_ACTION
```

#### SmartLabRun.st
```iecst
ACTION smartLabWorkstationOperation:
	CASE cm.state OF
		0:
			cm.description := 'Setting parameters for the workstations'; // None right now

			// Function block reference information
			ShuttlesAtPositions_0.shuttleInfo := ADR(gAcp6DCtrl.Status.ShuttleInfo); // Maybe need to run FB?
			ShuttlesInRange_0.shuttleInfo := ADR(gAcp6DCtrl.Status.ShuttleInfo);
			ShuttlesInWorkstationBuffer_0.shuttleInfo := ADR(gAcp6DCtrl.Status.ShuttleInfo);
			MovementColumnSelection_0.occupiedPosition := ADR(occupiedPosition);

			cm.state := 10;

		10:
			cm.description := 'Check what shuttle is on top of workstation';

			// Workstation position
			ShuttlesAtPositions_0.checkPosX[0] := pWorkstation.par.xLocation;
			ShuttlesAtPositions_0.checkPosY[0] := pWorkstation.par.yLocation;
			ShuttlesAtPositions_0.opt_checkShuttleState[0] := mcACP6D_SH_STATE_IDLING;
			ShuttlesAtPositions_0.numCheckedPos := 1;
			ShuttlesAtPositions_0();

			// Check if a shuttle is on the workstation and it is idle (meaning not in motion)
			IF ShuttlesAtPositions_0.isAtCheckPos  THEN
				pWorkstation.par.tempShuttleID := ShuttlesAtPositions_0.shuttleID;
				gShuttles[pWorkstation.par.tempShuttleID].par.tempWorkstationID := pWorkstation.par.workstationID;

				// If the shuttle is active, perform the operation
				IF shuttlePlans[pWorkstation.par.tempShuttleID].isActive THEN
					cm.state := 20;
				// If the shuttle is not active, go to wait for either new order or another shuttle in buffer
				ELSE
					cm.state := 15;
				END_IF
			END_IF

		15:
			cm.description := 'Wait for other shuttle to arrive at approach point or shuttle at workstation becomes part of new order';

			// Check if the shuttle should become part of a new order
			IF pWorkstation.par.workstationID = 0 THEN
				// New order has been read and must begin execution
				IF remainingOrderAmount > 0 THEN
					shuttlePlans[pWorkstation.par.tempShuttleID].isActive := TRUE;
					shuttlePlans[pWorkstation.par.tempShuttleID].progressIndex := 0;
					shuttlePlans[pWorkstation.par.tempShuttleID].routingSheet := CreateRouteSheet_0.outputRouteSheet;
					shuttlePlans[pWorkstation.par.tempShuttleID].productOrder := productOrder;

					remainingOrderAmount := remainingOrderAmount - 1;
					cm.state := 20;
				ELSIF NOT bufferEmpty THEN
					// Go back to read new order in read state
					em.substate := 17015;
				END_IF
			END_IF

			// Move to next workstation if another shuttle has arrived in the buffer of the workstation
			CASE pWorkstation.par.workstationID OF // For different workstations, you should look at differen positions
				0: // See if more than 2 shuttles are in queue
					// Position where at least 3 shuttles are in queue
					ShuttlesAtPositions_0.checkPosX[0] := pWorkstation.par.approachPosX - 0.240;
					ShuttlesAtPositions_0.checkPosY[0] := pWorkstation.par.approachPosY;
					ShuttlesAtPositions_0.opt_checkShuttleState[0] := mcACP6D_SH_STATE_OBSTACLE;
					ShuttlesAtPositions_0.numCheckedPos := 1;
					ShuttlesAtPositions_0();

					IF ShuttlesAtPositions_0.isAtCheckPos THEN
						// Set shuttle state to move to next workstation and go back to wait for new shuttle at workstation
						gShuttles[pWorkstation.par.tempShuttleID].cm.state := 10;
						cm.state := 60;
					END_IF

				1..5: // See if any shuttles are in the buffer
					ShuttlesInWorkstationBuffer_0.workstation := pWorkstation;
					ShuttlesInWorkstationBuffer_0();

					IF ShuttlesInWorkstationBuffer_0.isInBuffer THEN
						// Set shuttle state to move to next workstation and go back to wait for new shuttle at workstation
						gShuttles[pWorkstation.par.tempShuttleID].cm.state := 10;
						cm.state := 60;
					END_IF

			END_CASE

		20:
			cm.description := 'Send data to robot through mapping and begin robot operation';

			IF NOT robotBusy[i] THEN
				CASE pWorkstation.par.workstationID OF
					// Send type of bottom cover (converted to int)
					0: orderSpec[0] := COVER_TYPE_TO_USINT(shuttlePlans[pWorkstation.par.tempShuttleID].productOrder.bottomCover);

					// Send amount of holes
					1: orderSpec[1] := shuttlePlans[pWorkstation.par.tempShuttleID].productOrder.Holes;

					// Send whether a PCB is specified or not (converted to int)
					2: orderSpec[2] := BOOL_TO_USINT(shuttlePlans[pWorkstation.par.tempShuttleID].productOrder.PCB);

					// Send amount of fuses
					3: orderSpec[3] := shuttlePlans[pWorkstation.par.tempShuttleID].productOrder.Fuses;

					// Send type of top cover (converted to int)
					4: orderSpec[4] := COVER_TYPE_TO_USINT(shuttlePlans[pWorkstation.par.tempShuttleID].productOrder.topCover);

					// Send ID of order
					5:
						orderSpec[5] := shuttlePlans[pWorkstation.par.tempShuttleID].productOrder.ID;
						orderAmount := shuttlePlans[pWorkstation.par.tempShuttleID].productOrder.amount;

				END_CASE

				// Begin robot operation
				robotExecute[i] := TRUE;
				robotExecute[5] := FALSE; // To avoid robot 1 and 5 moving

				IF pWorkstation.par.landBeforeProcess THEN
					cm.state := 30;
				ELSE
					cm.state := 40;
				END_IF
			END_IF

		30:
			cm.description := 'Land shuttle if required';
			IF gAcp6DCtrl.Status.ShuttleInfo[pWorkstation.par.tempShuttleID].State = mcACP6D_SH_STATE_IDLING THEN
				pWorkstation.MC_BR_ShLevitation_Acp6D_0.Shuttle := ADR(gAcp6DCtrl.Status.ShuttleInfo[pWorkstation.par.tempShuttleID].shuttleRef);
				pWorkstation.MC_BR_ShLevitation_Acp6D_0.Parameters.Level := 0; //Land
				pWorkstation.MC_BR_ShLevitation_Acp6D_0.Parameters.Speed := 0;
				pWorkstation.MC_BR_ShLevitation_Acp6D_0.Execute := TRUE;
			END_IF
			IF pWorkstation.MC_BR_ShLevitation_Acp6D_0.Done THEN
				pWorkstation.MC_BR_ShLevitation_Acp6D_0.Execute := FALSE;
				cm.state := 40;
			END_IF

		40:
			cm.description := 'Wait for robot to finish operation';
			IF robotDone[i] THEN
				robotExecute[i] := FALSE;
				IF pWorkstation.par.landBeforeProcess THEN
					cm.state := 50;
				ELSE
					// Make current shuttle move to the next workstation and make workstation go back to wait for new shuttle
					gShuttles[pWorkstation.par.tempShuttleID].cm.state := 10;
					cm.state := 60;
				END_IF
			END_IF

		50:
			cm.description := 'Leviate shuttle if landed before process';
			pWorkstation.MC_BR_ShLevitation_Acp6D_0.Shuttle := ADR(gAcp6DCtrl.Status.ShuttleInfo[pWorkstation.par.tempShuttleID].shuttleRef);
			pWorkstation.MC_BR_ShLevitation_Acp6D_0.Parameters.Level := 1; //Leviate
			pWorkstation.MC_BR_ShLevitation_Acp6D_0.Parameters.Speed := 0;
			pWorkstation.MC_BR_ShLevitation_Acp6D_0.Execute := TRUE;
			IF pWorkstation.MC_BR_ShLevitation_Acp6D_0.Done THEN
				pWorkstation.MC_BR_ShLevitation_Acp6D_0.Execute := FALSE;

				gShuttles[pWorkstation.par.tempShuttleID].cm.state := 10;
				cm.state := 60;
			END_IF

		60:
			// Go back to wait for shuttle at workstation if the current shuttle has begun moving (avoids bugs)
			IF gAcp6DCtrl.Status.ShuttleInfo[pWorkstation.par.tempShuttleID].State = mcACP6D_SH_STATE_MOTION THEN
				cm.state := 10;
			END_IF

	END_CASE

	// Function block calls
	pWorkstation.MC_BR_ShLevitation_Acp6D_0();
	pWorkstation.TON_0();
	cm();

END_ACTION

ACTION smartLabShuttleMovement:

	CASE cm.state OF
		0:
			cm.description := 'Set parameters for the shuttles and wait for workstation to set new state';
			pShuttle.function.MC_BR_MoveInPlane_Acp6D_0.Parameters.Velocity := gAcp6DCtrl.Par.Velocity;
			pShuttle.function.MC_BR_MoveInPlane_Acp6D_0.Parameters.Acceleration := gAcp6DCtrl.Par.Acceleration;
			pShuttle.function.MC_BR_MoveInPlane_Acp6D_0.Parameters.Mode := 0; //Absolute

		10:
			cm.description := 'Determine where to move next';

			// Set the next workstation ID (either from routing sheet for active shuttles and next in row for inactive shuttles)
			IF pShuttlePlan.isActive THEN
				pShuttle.par.tempNextWorkstationID := pShuttlePlan.routingSheet[pShuttlePlan.progressIndex];

				// If the next workstation is 0 reset the progress index and set the shuttleplan to be inactive, otherwise increment progress index by 1
				IF pShuttlePlan.routingSheet[pShuttlePlan.progressIndex] = 0 THEN
					pShuttlePlan.progressIndex := 0;
					pShuttlePlan.isActive := FALSE;
					activeShuttles := activeShuttles - 1;
				ELSE
					pShuttlePlan.progressIndex := pShuttlePlan.progressIndex + 1;
				END_IF
			ELSE
				pShuttle.par.tempNextWorkstationID := (pShuttle.par.tempWorkstationID + 1) MOD smartLabNumWorkstations;
			END_IF

			// If the workstations are opposite each other, go directly to the approach point of next workstation (no need to occupy column when it only moves in row)
			IF AreWorkstationsOpposite(workstationID1 := pShuttle.par.tempWorkstationID, workstationID2 := pShuttle.par.tempNextWorkstationID) THEN
				cm.state := 30;
			// If the workstations are adjacent to each other and the buffer to the next workstation is empty, move directly to the workstation
			ELSIF AreWorkstationsAdjacent(workstationID1 := pShuttle.par.tempWorkstationID, workstationID2 := pShuttle.par.tempNextWorkstationID) THEN
				// Define the next workstation
				ShuttlesInWorkstationBuffer_0.workstation := gWorkstations[pShuttle.par.tempNextWorkstationID];
				ShuttlesInWorkstationBuffer_0();

				IF ShuttlesInWorkstationBuffer_0.isInBuffer THEN
					cm.state := 20;
				ELSE
					cm.state := 40;
				END_IF
			// Else move using original method (find free column to use)
			ELSE
				cm.state := 20;
			END_IF

		20:
			cm.description := 'Move from workstation to depart point (or next free column)';
			pShuttle.function.MC_BR_MoveInPlane_Acp6D_0.Shuttle := ADR(gAcp6DCtrl.Status.ShuttleInfo[pShuttle.par.shuttleID].shuttleRef);
			pShuttle.function.MC_BR_MoveInPlane_Acp6D_0.Parameters.Path := 2; // Y THEN X

			// If a column has not been selected yet
			IF pShuttle.par.tempHighwayColumn = -1 THEN
				// Select the closest column that is available (no other shuttles using column or movement direction is opposite)
				MovementColumnSelection_0.startWorkstation := gWorkstations[pShuttle.par.tempWorkstationID];
				MovementColumnSelection_0.endWorkstation := gWorkstations[pShuttle.par.tempNextWorkstationID];
				MovementColumnSelection_0();

				pShuttle.par.tempHighwayColumn := MovementColumnSelection_0.selectedColumn;

			// Move to the specified column if any is available (-1 if no column is available)
			ELSE
				// Position of the selected column
				pShuttle.function.MC_BR_MoveInPlane_Acp6D_0.Parameters.Position.X := QuadrantIdxToPos(quadrantIdx := (1 + pShuttle.par.tempHighwayColumn)); // Add 1 because the first column is not a highway
				pShuttle.function.MC_BR_MoveInPlane_Acp6D_0.Parameters.Position.Y := gWorkstations[pShuttle.par.tempWorkstationID].par.departPosY;

				pShuttle.function.MC_BR_MoveInPlane_Acp6D_0.Execute := TRUE;
				IF pShuttle.function.MC_BR_MoveInPlane_Acp6D_0.Done THEN
					pShuttle.function.MC_BR_MoveInPlane_Acp6D_0.Execute := FALSE;

					cm.state := 30;
				END_IF
			END_IF

		30:
			cm.description := 'Move from depart point (or free row) of current workstation to approach point of next workstation';
			pShuttle.function.MC_BR_MoveInPlane_Acp6D_0.Shuttle := ADR(gAcp6DCtrl.Status.ShuttleInfo[pShuttle.par.shuttleID].shuttleRef);
			pShuttle.function.MC_BR_MoveInPlane_Acp6D_0.Parameters.Path := 2; // Y THEN X

			// Move to approach point of next workstation specified in the routing sheet (or just the next workstation if the shuttle is inactive)
			pShuttle.function.MC_BR_MoveInPlane_Acp6D_0.Parameters.Position.X := gWorkstations[pShuttle.par.tempNextWorkstationID].par.approachPosX;
			pShuttle.function.MC_BR_MoveInPlane_Acp6D_0.Parameters.Position.Y := gWorkstations[pShuttle.par.tempNextWorkstationID].par.approachPosY;

			pShuttle.function.MC_BR_MoveInPlane_Acp6D_0.Execute := TRUE;
			IF pShuttle.function.MC_BR_MoveInPlane_Acp6D_0.Done THEN
				pShuttle.function.MC_BR_MoveInPlane_Acp6D_0.Execute := FALSE;

				// Make the positions available for use again if any were occupied by the movement
				IF NOT AreWorkstationsOpposite(workstationID1 := pShuttle.par.tempWorkstationID, workstationID2 := pShuttle.par.tempNextWorkstationID) THEN
					MovementColumnSelection_0.startWorkstation := gWorkstations[pShuttle.par.tempWorkstationID];
					MovementColumnSelection_0.endWorkstation := gWorkstations[pShuttle.par.tempNextWorkstationID];
					MovementColumnSelection_0.opt_movementDone := TRUE;
					MovementColumnSelection_0.opt_resetColumn := pShuttle.par.tempHighwayColumn;
					MovementColumnSelection_0();

					pShuttle.par.tempHighwayColumn := -1;
				END_IF

				cm.state := 40;
			END_IF

		40:
			cm.description := 'Move from approach point to workstation';
			pShuttle.function.MC_BR_MoveInPlane_Acp6D_0.Shuttle := ADR(gAcp6DCtrl.Status.ShuttleInfo[pShuttle.par.shuttleID].shuttleRef);
			pShuttle.function.MC_BR_MoveInPlane_Acp6D_0.Parameters.Path := 1; // X THEN Y

			// Move to next workstation
			pShuttle.function.MC_BR_MoveInPlane_Acp6D_0.Parameters.Position.X := gWorkstations[pShuttle.par.tempNextWorkstationID].par.xLocation;
			pShuttle.function.MC_BR_MoveInPlane_Acp6D_0.Parameters.Position.Y := gWorkstations[pShuttle.par.tempNextWorkstationID].par.yLocation;

			pShuttle.function.MC_BR_MoveInPlane_Acp6D_0.Execute := TRUE;
			IF pShuttle.function.MC_BR_MoveInPlane_Acp6D_0.Acknowledge THEN
				pShuttle.function.MC_BR_MoveInPlane_Acp6D_0.Execute := FALSE;

				// Go back to wait for new workstation to send the shuttle on
				cm.state := 0;
			END_IF

	END_CASE

	// Function block calls
	pShuttle.function.MC_BR_MoveInPlane_Acp6D_0();
	cm();

END_ACTION
```

#### Types.typ - Local data types
```iecst
TYPE
	shuttle_plan : 	STRUCT
		productOrder : product_order;
		routingSheet : ARRAY[0..5]OF USINT;
		progressIndex : USINT := 0;
		isActive : BOOL;
	END_STRUCT;
	shuttle_status_typ : 	STRUCT
		dummy : USINT;
	END_STRUCT;
	shuttle_par_typ : 	STRUCT
		shuttleID : USINT;
		tempWorkstationID : USINT;
		tempNextWorkstationID : USINT;
		tempHighwayColumn : SINT;
	END_STRUCT;
	shuttle_function_typ : 	STRUCT
		MC_BR_Move6D_Acp6D_0 : MC_BR_Move6D_Acp6D;
		MC_BR_MoveShortAxis_Acp6D_0 : MC_BR_MoveShortAxis_Acp6D;
		MC_BR_ShGetPayload_Acp6D_0 : MC_BR_ShGetPayload_Acp6D;
		MC_BR_MoveInPlane_Acp6D_0 : MC_BR_MoveInPlane_Acp6D;
		TON_0 : TON;
	END_STRUCT;
	shuttlePos : 	STRUCT
		xPos : REAL;
		yPos : REAL;
	END_STRUCT;
	test_typ : 	STRUCT
		targetReached : ARRAY[0..3]OF BOOL := [4(FALSE)];
	END_STRUCT;
	thisShuttleSetup : 	STRUCT
		Shuttle2 : shuttlePos;
		Shuttle3 : shuttlePos;
		Shuttle4 : shuttlePos;
		Shuttle1 : shuttlePos;
	END_STRUCT;
	ABB_typ : 	STRUCT
		HomePositionReached : BOOL;
		startSmallWeightMovement : BOOL;
		returnBigWeightMovement : BOOL;
		returnSmallWeightMovement : BOOL;
		startBigWeightMovement : BOOL;
	END_STRUCT;
	shuttle_typ : 	STRUCT
		cm : brdkCM;
		status : shuttle_status_typ;
		par : shuttle_par_typ;
		function : shuttle_function_typ;
	END_STRUCT;
	workStation_cmd_typ : 	STRUCT
		dummy : USINT;
	END_STRUCT;
	workStation_par_typ : 	STRUCT
		landBeforeProcess : BOOL; (*TRUE = yes*)
		yLocation : REAL;
		xLocation : REAL;
		tempShuttleID : USINT;
		workstationID : USINT;
		nextStationSelector : STRING[10];
		processTime : REAL;
		pathRouting : USINT := 0; (*0 Diagonal, 1 First X then Y, 2 First Y then X*)
		ArcMovement : BOOL;
		approachPosX : REAL;
		approachPosY : REAL;
		departPosX : REAL;
		departPosY : REAL;
	END_STRUCT;
	workStation_status_typ : 	STRUCT
		componentName : STRING[80];
		active : BOOL;
		oneshot : BOOL;
	END_STRUCT;
	workStation_typ : 	STRUCT
		par : workStation_par_typ;
		status : workStation_status_typ;
		cmd : workStation_cmd_typ;
		cm : brdkCM;
		MC_BR_RotaryMotionSpin_Acp6D_0 : MC_BR_RotaryMotionSpin_Acp6D;
		MC_BR_RotaryMotion_Acp6D_0 : MC_BR_RotaryMotion_Acp6D;
		MC_BR_MoveInPlane_Acp6D_0 : MC_BR_MoveInPlane_Acp6D;
		MC_BR_ShLevitation_Acp6D_0 : MC_BR_ShLevitation_Acp6D;
		TON_0 : TON;
		workstationSwitcher : BOOL;
		MC_BR_MoveArc_Acp6D_0 : MC_BR_MoveArc_Acp6D;
		MC_BR_Move6D_Acp6D_0 : MC_BR_Move6D_Acp6D;
	END_STRUCT;
	product_order : 	STRUCT
		amount : USINT;
		bottomCover : cover_types;
		Holes : USINT;
		PCB : BOOL;
		Fuses : USINT;
		topCover : cover_types;
		ID : USINT;
	END_STRUCT;
	cover_types :
		(
		noCover := 0,
		blackCover := 1,
		whiteCover := 2,
		blueCover := 3
		);
END_TYPE
```

#### Variables.var - Local variables
```iecst
VAR
	ABBRobot : ABB_typ;
	cm : REFERENCE TO brdkCM;
	createShGroup : USINT;
	em : brdkEM;
	enableButtons : BOOL;
	fbPayload : REAL;
	flaskProgramAcceleration : REAL := 0.2;
	flaskProgramVelocity : REAL := 2;
	gShuttles : ARRAY[0..NUM_SHUTTLES] OF shuttle_typ;
	gWorkstations : ARRAY[0..NR_OF_WORKSTATIONS] OF workStation_typ;
	i : USINT;
	j : USINT;
	k : USINT;
	localCurrentNumShuttles : UINT;
	macroCreater : USINT;
	MARGIN : REAL := 0.0059;
	MC_BR_AsmGetInfo_Acp6D_0 : MC_BR_AsmGetInfo_Acp6D;
	MC_BR_AsmGetShuttle_Acp6D_0 : MC_BR_AsmGetShuttle_Acp6D;
	MC_BR_AsmLevitation_Acp6D_0 : MC_BR_AsmLevitation_Acp6D;
	MC_BR_AsmPowerOff_Acp6D_0 : MC_BR_AsmPowerOff_Acp6D;
	MC_BR_AsmPowerOn_Acp6D_0 : MC_BR_AsmPowerOn_Acp6D;
	MC_BR_AsmReadStatus_Acp6D_0 : MC_BR_AsmReadStatus_Acp6D;
	MC_BR_AsmStop_Acp6D_0 : MC_BR_AsmStop_Acp6D;
	MC_BR_MacroCreate_Acp6D_0 : MC_BR_MacroCreate_Acp6D;
	MC_BR_MacroRun_Acp6D_0 : MC_BR_MacroRun_Acp6D;
	MC_BR_MacroSave_Acp6D_0 : MC_BR_MacroSave_Acp6D;
	MC_BR_Move6D_Acp6D_0 : MC_BR_Move6D_Acp6D;
	MC_BR_MoveArc_Acp6D_0 : MC_BR_MoveArc_Acp6D;
	MC_BR_MoveInPlaneAsync_Acp6D_0 : MC_BR_MoveInPlaneAsync_Acp6D;
	MC_BR_MoveInPlane_Acp6D_0 : MC_BR_MoveInPlane_Acp6D;
	MC_BR_MoveShortAxis_Acp6D_0 : ARRAY[0..3] OF MC_BR_MoveShortAxis_Acp6D;
	MC_BR_ReadCyclicPosition_Acp6D_0 : MC_BR_ReadCyclicPosition_Acp6D;
	MC_BR_ReadCyclicPosition_Acp6D_1 : MC_BR_ReadCyclicPosition_Acp6D;
	MC_BR_ReadCyclicPosition_Acp6D_2 : MC_BR_ReadCyclicPosition_Acp6D;
	MC_BR_ReadCyclicPosition_Acp6D_3 : MC_BR_ReadCyclicPosition_Acp6D;
	MC_BR_RotaryMotionSpin_Acp6D_0 : MC_BR_RotaryMotionSpin_Acp6D;
	MC_BR_RotaryMotion_Acp6D_0 : MC_BR_RotaryMotion_Acp6D;
	MC_BR_ShGroupAddShuttle_Acp6D_0 : MC_BR_ShGroupAddShuttle_Acp6D;
	MC_BR_ShGroupCoupleCtrl_Acp6D_0 : MC_BR_ShGroupCoupleCtrl_Acp6D;
	MC_BR_ShGroupCreate_Acp6D_0 : MC_BR_ShGroupCreate_Acp6D;
	MC_BR_ShGroupCreate_Acp6D_1 : MC_BR_ShGroupCreate_Acp6D;
	MC_BR_ShGroupCreate_Acp6D_2 : MC_BR_ShGroupCreate_Acp6D;
	MC_BR_ShGroupCreate_Acp6D_3 : MC_BR_ShGroupCreate_Acp6D;
	MC_BR_ShGroupCreate_Acp6D_4 : MC_BR_ShGroupCreate_Acp6D;
	MC_BR_ShGroupGetInfo_Acp6D_0 : MC_BR_ShGroupGetInfo_Acp6D;
	MC_BR_ShLevitation_Acp6D_0 : MC_BR_ShLevitation_Acp6D;
	MC_BR_ShReadInfo_Acp6D_0 : ARRAY[0..NUM_SHUTTLES] OF MC_BR_ShReadInfo_Acp6D;
	positionContainerBoxProgram : ARRAY[0..9] OF shuttleStartup_typ;
	positionContainerFlaskProgram : ARRAY[0..9] OF shuttleStartup_typ;
	positionContainerLinkMovement : ARRAY[0..7] OF thisShuttleSetup;
	positionContainerLinkMovementNew : ARRAY[0..9] OF shuttleStartup_typ;
	positionContainerRotation : ARRAY[0..9] OF shuttleStartup_typ;
	positionContainerSteelSheet : ARRAY[0..9] OF shuttleStartup_typ;
	positionContainerTestProgram : ARRAY[0..7] OF shuttleStartup_typ;
	positionContainerWorkstationMov : ARRAY[0..9] OF shuttleStartup_typ;
	shGroupShuttle1_2 : UDINT;
	shGroupShuttle1_4 : UDINT;
	shGroupShuttle2_3 : UDINT;
	shGroupShuttle3_4 : UDINT;
	shGroupShuttle5_6_7_8 : UDINT;
	shuttlePayload : REAL;
	shuttleToTakePictureOf : USINT;
	steelSheetFlyingHeight : REAL := 0.002;
	tempCounter : USINT;
	tempShuttleCnt : USINT;
	tempShuttleCounter : USINT;
	testObj : test_typ;
	TON_watchdog : TON;
	weightCalibration : REAL;
END_VAR
VAR RETAIN
	weightProgramFlyingHight : REAL := 1.3;
END_VAR
(*-----------------------------------*)
(*////////// SMART LAB \\\\\\\\\\*)
(*-----------------------------------*)
VAR
	activeShuttles : USINT;
	amountProductsFinished : USINT;
	availablePosition : {REDUND_UNREPLICABLE} ARRAY[0..3,0..7] OF BOOL; (*4 highway columns and 8 highway rows*)
	bufferEmpty : BOOL := TRUE;
	bufferFull : BOOL := FALSE;
	bufferSize : {REDUND_UNREPLICABLE} USINT;
	MovementColumnSelection_0 : MovementColumnSelection;
	CreateRouteSheet_0 : {REDUND_UNREPLICABLE} CreateRouteSheet;
	executeOrder : BOOL := FALSE;
	orderBuffer : ARRAY[0..9] OF product_order := [10((amount:=0,bottomCover:=noCover,topCover:=noCover,PCB:=FALSE,Fuses:=0,ID:=0))];
	positionContainerSmartLabProgram : ARRAY[0..7] OF shuttleStartup_typ;
	productOrder : product_order := (amount:=1,topCover:=blackCover,bottomCover:=blackCover,PCB:=TRUE,Fuses:=2);
	pShuttle : REFERENCE TO shuttle_typ;
	pShuttlePlan : REFERENCE TO shuttle_plan;
	pWorkstation : REFERENCE TO workStation_typ;
	remainingOrderAmount : USINT;
	ShuttlesAtPositions_0 : ShuttlesAtPositions;
	ShuttlesInRange_0 : ShuttlesInRange;
	ShuttlesInWorkstationBuffer_0 : ShuttlesInWorkstationBuffer;
	shuttlePlans : ARRAY[0..7] OF shuttle_plan;
END_VAR
VAR CONSTANT
	smartLabNumShuttles : USINT := 8;
	smartLabNumWorkstations : USINT := 6;
END_VAR
VAR
	tempProductOrder : product_order := (amount:=1,bottomCover:=blackCover,topCover:=blackCover,PCB:=TRUE,Fuses:=2,Holes:=4);
	tempShuttleIndex : USINT;
	TON_0 : TON;
	readIndex : USINT := 0;
	writeIndex : USINT := 0;
END_VAR
(*Variable mapping*)
VAR
	orderSpec : ARRAY[0..5] OF SINT;
	orderAmount : SINT;
	robotExecute : ARRAY[0..5] OF BOOL;
	robotDone : ARRAY[0..5] OF BOOL;
	robotBusy : ARRAY[0..5] OF BOOL;
END_VAR
```

#### LocalFunctions.fun
```iecst
{REDUND_OK} FUNCTION_BLOCK CreateRouteSheet (*TODO: Add your comment here*) (*$GROUP=User,$CAT=User,$GROUPICON=User.png,$CATICON=User.png*)
	VAR_INPUT
		inputProductOrder : product_order;
	END_VAR
	VAR_OUTPUT
		outputRouteSheet : ARRAY[0..5] OF USINT;
	END_VAR
	VAR
		i : USINT;
		tempIndex : USINT;
		routeSize : USINT;
	END_VAR
END_FUNCTION_BLOCK

{REDUND_ERROR} FUNCTION_BLOCK MovementColumnSelection
	VAR_INPUT
		availablePosition : REFERENCE TO ARRAY[0..3,0..7] OF BOOL; (*4 highway columns and 8 highway rows*)
		startWorkstation : workStation_typ;
		endWorkstation : workStation_typ;
		opt_movementDone : BOOL; (*Reset the positions that were occupied by the movement*)
		opt_resetColumn : SINT;
	END_VAR
	VAR_OUTPUT
		selectedColumn : SINT;
	END_VAR
	VAR
		startRowLevel : USINT;
		endRowLevel : USINT;
		columnIsPossible : BOOL;
		i : USINT;
		k : USINT;
	END_VAR
END_FUNCTION_BLOCK

{REDUND_ERROR} FUNCTION_BLOCK ShuttlesAtPositions (*TODO: Add your comment here*) (*$GROUP=User,$CAT=User,$GROUPICON=User.png,$CATICON=User.png*)
	VAR_INPUT
		shuttleInfo : REFERENCE TO ARRAY[0..NUM_SHUTTLES] OF ShuttleInfoType;
		checkPosX : ARRAY[0..7] OF REAL; (*Should technically be 48 (12 segments * 4 positions)*)
		checkPosY : ARRAY[0..7] OF REAL; (*Should technically be 48 (12 segments * 4 positions)*)
		opt_checkShuttleState : ARRAY[0..7] OF McAcp6DShStateEnum := [8(0)]; (*Don't set if all states should be checked*)
		numCheckedPos : USINT;
	END_VAR
	VAR_OUTPUT
		isAtCheckPos : BOOL;
		shuttleID : USINT;
	END_VAR
	VAR
		i : USINT;
		k : USINT;
		MARGIN : REAL := 0.005;
		numShuttles : USINT := 8;
	END_VAR
END_FUNCTION_BLOCK

{REDUND_ERROR} FUNCTION_BLOCK ShuttlesInRange
	VAR_INPUT
		shuttleInfo : REFERENCE TO ARRAY[0..NUM_SHUTTLES] OF ShuttleInfoType;
		checkRangeX1 : REAL;
		checkRangeX2 : REAL;
		checkRangeY1 : REAL;
		checkRangeY2 : REAL;
	END_VAR
	VAR_OUTPUT
		isInRange : BOOL;
	END_VAR
	VAR
		checkRangeStartX : REAL;
		checkRangeEndX : REAL;
		checkRangeStartY : REAL;
		checkRangeEndY : REAL;
		i : USINT;
	END_VAR
	VAR CONSTANT
		MARGIN : REAL := 0.005;
		numShuttles : USINT := 8;
	END_VAR
END_FUNCTION_BLOCK

FUNCTION_BLOCK ShuttlesInWorkstationBuffer
	VAR_INPUT
		shuttleInfo : REFERENCE TO ARRAY[0..NUM_SHUTTLES] OF ShuttleInfoType;
		workstation : workStation_typ;
	END_VAR
	VAR_OUTPUT
		isInBuffer : BOOL;
	END_VAR
	VAR
		ShuttlesAtPositions_0 : ShuttlesAtPositions;
		ShuttlesInRange_0 : ShuttlesInRange;
	END_VAR
	VAR CONSTANT
		MARGIN : REAL := 0.005;
	END_VAR
END_FUNCTION_BLOCK

{REDUND_ERROR} FUNCTION AreWorkstationsOpposite : BOOL (* *) (*$GROUP=User,$CAT=User,$GROUPICON=User.png,$CATICON=User.png*)
	VAR_INPUT
		workstationID1 : INT;
		workstationID2 : INT;
	END_VAR
END_FUNCTION

{REDUND_ERROR} FUNCTION AreWorkstationsAdjacent : BOOL
	VAR_INPUT
		workstationID1 : INT;
		workstationID2 : INT;
	END_VAR
END_FUNCTION

{REDUND_ERROR} FUNCTION QuadrantIdxToPos : REAL
	VAR_INPUT
		quadrantIdx : USINT;
	END_VAR
END_FUNCTION

FUNCTION PosToQuadrantIdx : USINT
	VAR_INPUT
		pos : REAL;
	END_VAR
END_FUNCTION

{REDUND_ERROR} FUNCTION COVER_TYPE_TO_USINT : USINT (*TODO: Add your comment here*) (*$GROUP=User,$CAT=User,$GROUPICON=User.png,$CATICON=User.png*)
	VAR_INPUT
		coverType : cover_types;
	END_VAR
END_FUNCTION
```

#### createRouteSheet.st
```iecst
(* TODO: Add your comment here *)
FUNCTION_BLOCK CreateRouteSheet

	routeSize := SIZEOF(outputRouteSheet)/SIZEOF(outputRouteSheet[0]);
	tempIndex := 0;

	FOR i := 0 TO routeSize DO
		outputRouteSheet[i] := 0;
	END_FOR

	// Check if visitation to drilling station is required
	IF inputProductOrder.Holes <> 0 THEN

		outputRouteSheet[tempIndex] := 1; // WORKSTATION 1
		tempIndex := tempIndex + 1;

	END_IF

	// Check if visitation to PCB station is required
	IF inputProductOrder.PCB THEN

		outputRouteSheet[tempIndex] := 2; // WORKSTATION 2
		tempIndex := tempIndex + 1;

		// Check if visitation to fuse station is required
		IF inputProductOrder.Fuses > 0 THEN

			outputRouteSheet[tempIndex] := 3; // WORKSTATION 3
			tempIndex := tempIndex + 1;

		END_IF

	END_IF

	// Check if visitation to top cover station is required
	IF inputProductOrder.topCover <> noCover THEN

		outputRouteSheet[tempIndex] := 4; // WORKSTATION 4
		tempIndex := tempIndex + 1;

	END_IF

	// The order is unloaded
	outputRouteSheet[tempIndex] := 5; // WORKSTATION 5

END_FUNCTION_BLOCK
```

#### quadrantIdxToPos.st
```iecst
(* TODO: Add your comment here *)
FUNCTION QuadrantIdxToPos

	QuadrantIdxToPos := quadrantIdx*0.120 + 0.060;

END_FUNCTION
```

#### COVER_TYPE_TO_USINT.st
```iecst
(* TODO: Add your comment here *)
FUNCTION COVER_TYPE_TO_USINT

	CASE coverType OF

		noCover:

			COVER_TYPE_TO_USINT := 0;

		blackCover:

			COVER_TYPE_TO_USINT := 1;

		whiteCover:

			COVER_TYPE_TO_USINT := 2;

		blueCover:

			COVER_TYPE_TO_USINT := 3;

	END_CASE

END_FUNCTION
```

#### ShuttlesAt.st
```iecst
FUNCTION_BLOCK ShuttlesAtPositions

	// Access the shuttle information
	shuttleInfo ACCESS ADR(shuttleInfo);

	// Shuttle is not at checkPos by default
	isAtCheckPos := FALSE;

	// Check if a shuttle is at any of the positions
	FOR k := 0 TO (numCheckedPos - 1) DO
		FOR i := 0 TO (numShuttles - 1) DO
			IF ((shuttleInfo[i].Position.X > checkPosX[k] - MARGIN AND shuttleInfo[i].Position.X < checkPosX[k] + MARGIN) AND
				(shuttleInfo[i].Position.Y > checkPosY[k] - MARGIN AND shuttleInfo[i].Position.Y < checkPosY[k] + MARGIN)) AND
				(opt_checkShuttleState[k] = 0 OR shuttleInfo[i].State = opt_checkShuttleState[k]) THEN // Shuttle state 0 corresponds to any state being accepted
				isAtCheckPos := TRUE;
				shuttleID := i;
				EXIT;
			END_IF
		END_FOR

		IF isAtCheckPos THEN
			 // Done such that shuttleID will be the first checked position with shuttle (in case there are shuttles at several of the checked positions)
			EXIT;
		END_IF
	END_FOR

	// Reset checkShuttleState for next time FB is called
	FOR k := 0 TO (numCheckedPos - 1) DO
		opt_checkShuttleState[k] := 0;
	END_FOR

END_FUNCTION_BLOCK

FUNCTION_BLOCK ShuttlesInRange

	// Access the shuttle information
	shuttleInfo ACCESS ADR(shuttleInfo);

	// Setting start and end range of X
	IF checkRangeX1 < checkRangeX2 THEN
		checkRangeStartX := checkRangeX1;
		checkRangeEndX := checkRangeX2;
	ELSE
		checkRangeStartX := checkRangeX2;
		checkRangeEndX := checkRangeX1;
	END_IF

	// Setting start and end range of Y
	IF checkRangeY1 < checkRangeY2 THEN
		checkRangeStartY := checkRangeY1;
		checkRangeEndY := checkRangeY2;
	ELSE
		checkRangeStartY := checkRangeY2;
		checkRangeEndY := checkRangeY1;
	END_IF

	// Shuttle is not in the range by default
	isInRange := FALSE;

	// Check if the shuttle is in the rectangular range
	FOR i := 0 TO (numShuttles - 1) DO
		IF (shuttleInfo[i].Position.X > checkRangeStartX - MARGIN AND shuttleInfo[i].Position.X < checkRangeEndX + MARGIN) AND
			(shuttleInfo[i].Position.Y > checkRangeStartY - MARGIN AND shuttleInfo[i].Position.Y < checkRangeEndY + MARGIN) THEN
			isInRange := TRUE;
			EXIT;
		END_IF
	END_FOR

END_FUNCTION_BLOCK

FUNCTION_BLOCK ShuttlesInWorkstationBuffer

	// Access the shuttle information
	shuttleInfo ACCESS ADR(shuttleInfo);

	// Set the address of shuttleinfo to the function blocks
	ShuttlesAtPositions_0.shuttleInfo := ADR(shuttleInfo);
	ShuttlesInRange_0.shuttleInfo := ADR(shuttleInfo);

	// Shuttle is not in the buffer by default
	isInBuffer := FALSE;

	// Check idle shuttle at approach point
	ShuttlesAtPositions_0.checkPosX[0] := workstation.par.approachPosX;
	ShuttlesAtPositions_0.checkPosY[0] := workstation.par.approachPosY;
	ShuttlesAtPositions_0.opt_checkShuttleState[0] := mcACP6D_SH_STATE_IDLING;
	ShuttlesAtPositions_0.numCheckedPos := 1;
	ShuttlesAtPositions_0();

	// Check rest of buffer
	IF workstation.par.workstationID <= 2 THEN
		ShuttlesInRange_0.checkRangeX1 := workstation.par.approachPosX + 2*MARGIN; // 2*MARGIN to avoid checking approach point
	ELSE
		ShuttlesInRange_0.checkRangeX1 := workstation.par.approachPosX - 2*MARGIN;
	END_IF
	ShuttlesInRange_0.checkRangeX2 := workstation.par.xLocation;
	ShuttlesInRange_0.checkRangeY1 := workstation.par.approachPosY;
	ShuttlesInRange_0.checkRangeY2 := workstation.par.approachPosY;
	ShuttlesInRange_0();

	IF ShuttlesAtPositions_0.isAtCheckPos OR ShuttlesInRange_0.isInRange THEN
		isInBuffer := TRUE;
	END_IF

END_FUNCTION_BLOCK
```

#### Conversions.st - not listed in the package file held
```iecst
// Quadrant index to meter position conversion
FUNCTION QuadrantIdxToPos

	QuadrantIdxToPos := quadrantIdx*0.120 + 0.060;

END_FUNCTION

FUNCTION PosToQuadrantIdx

	PosToQuadrantIdx := REAL_TO_USINT(brmfloor(pos) / 0.120);

END_FUNCTION

// Cover type to USINT conversion
FUNCTION COVER_TYPE_TO_USINT

	CASE coverType OF

		noCover:

			COVER_TYPE_TO_USINT := 0;

		blackCover:

			COVER_TYPE_TO_USINT := 1;

		whiteCover:

			COVER_TYPE_TO_USINT := 2;

		blueCover:

			COVER_TYPE_TO_USINT := 3;

	END_CASE

END_FUNCTION
```

#### Danfoss.st - not listed in the package file held
```iecst
ACTION danfossAction:
	//Setup
	positionDanfoss[0].initXPos											:= 0.430;
	positionDanfoss[0].initYPos											:= 0.420;
	positionDanfoss[1].initXPos											:= 0.420;
	positionDanfoss[1].initYPos											:= 0.300;
	positionDanfoss[2].initXPos											:= 0.430;
	positionDanfoss[2].initYPos											:= 0.180;
	positionDanfoss[3].initXPos											:= 0.420;
	positionDanfoss[3].initYPos											:= 0.060;

	gWorkStations[0].par.xLocation										:= 0.430;
	gWorkStations[0].par.yLocation										:= 0.180;
	gWorkStations[0].par.nextStationSelector							:= '1';
	gWorkStations[0].par.processTime									:= danfossWorkStation1Timer;
	gWorkStations[0].par.pathRouting									:= 1;
	gWorkStations[0].par.ArcMovement									:= FALSE;
	gWorkStations[0].par.landBeforeProcess								:= TRUE;
	gWorkStations[0].par.internalCounter								:= danfossWorkStation1NUMRotations;

	gWorkStations[1].par.xLocation										:= 0.430;
	gWorkStations[1].par.yLocation										:= 0.420;
	gWorkStations[1].par.nextStationSelector							:= '0';
	gWorkStations[1].par.processTime									:= danfossWorkStation2Timer;
	gWorkStations[1].par.pathRouting									:= 2;
	gWorkStations[1].par.ArcMovement									:= FALSE;
	gWorkStations[1].par.landBeforeProcess								:= TRUE;
	gWorkStations[1].par.internalCounter								:= danfossWorkStation2NUMRotations;

	gWorkStations[2].par.xLocation										:= 0.000;
	gWorkStations[2].par.yLocation										:= 0.000;
	gWorkStations[2].par.nextStationSelector							:= '0';
	gWorkStations[2].par.processTime									:= 0;
	gWorkStations[2].par.pathRouting									:= 0;
	gWorkStations[2].par.ArcMovement									:= FALSE;

	gWorkStations[3].par.xLocation										:= 0.000;
	gWorkStations[3].par.yLocation										:= 0.000;
	gWorkStations[3].par.nextStationSelector							:= '0';
	gWorkStations[3].par.processTime									:= 0;
	gWorkStations[3].par.pathRouting									:= 0;
	gWorkStations[3].par.ArcMovement									:= FALSE;

	//Setup WorkStations
	CASE em.substate OF
		10000:
			em.description := 'Move shuttle to pre pos';
			gWorkStations[1].status.oneshot := TRUE;
			tempShuttleCounter := 0;
			MC_BR_MoveInPlaneAsync_Acp6D_0.Parameters.Acceleration := gAcp6DCtrl.Par.Acceleration;
			MC_BR_MoveInPlaneAsync_Acp6D_0.Parameters.Velocity := gAcp6DCtrl.Par.Velocity;
			FOR i := 0 TO NUM_SHUTTLES DO
				MC_BR_MoveInPlaneAsync_Acp6D_0.Parameters.AsyncPar[i].Shuttle := ADR(gAcp6DCtrl.Status.ShuttleInfo[i].shuttleRef);
				MC_BR_MoveInPlaneAsync_Acp6D_0.Parameters.AsyncPar[i].X := positionDanfoss[i].initXPos;
				MC_BR_MoveInPlaneAsync_Acp6D_0.Parameters.AsyncPar[i].Y := positionDanfoss[i].initYPos;
			END_FOR;
			MC_BR_MoveInPlaneAsync_Acp6D_0.Execute := TRUE;
			IF MC_BR_MoveInPlaneAsync_Acp6D_0.Acknowledge THEN
				MC_BR_MoveInPlaneAsync_Acp6D_0.Execute := FALSE;
				em.substate := 10010;
			END_IF

		10010:
			em.description := 'Move shuttle 2 towards workstation 2';
			MC_BR_MoveInPlane_Acp6D_0.Parameters.Acceleration := gAcp6DCtrl.Par.Acceleration;
			MC_BR_MoveInPlane_Acp6D_0.Parameters.Velocity := gAcp6DCtrl.Par.Velocity;
			MC_BR_MoveInPlane_Acp6D_0.Shuttle := ADR(gAcp6DCtrl.Status.ShuttleInfo[1].shuttleRef);
			MC_BR_MoveInPlane_Acp6D_0.Parameters.Position.X := 0.420;
			MC_BR_MoveInPlane_Acp6D_0.Parameters.Position.Y := 0.420;
			MC_BR_MoveInPlane_Acp6D_0.Parameters.Path := 0;
			MC_BR_MoveInPlane_Acp6D_0.Parameters.Mode := 0;
			MC_BR_MoveInPlane_Acp6D_0.Execute := TRUE;
			IF MC_BR_MoveInPlane_Acp6D_0.Acknowledge THEN
				MC_BR_MoveInPlane_Acp6D_0.Execute := FALSE;
				em.substate := 10015;
			END_IF

		10015:
			em.description := 'Move shuttle 2 towards workstation 2';
			MC_BR_MoveInPlane_Acp6D_0.Parameters.Acceleration := gAcp6DCtrl.Par.Acceleration;
			MC_BR_MoveInPlane_Acp6D_0.Parameters.Velocity := gAcp6DCtrl.Par.Velocity;
			MC_BR_MoveInPlane_Acp6D_0.Shuttle := ADR(gAcp6DCtrl.Status.ShuttleInfo[1].shuttleRef);
			MC_BR_MoveInPlane_Acp6D_0.Parameters.Position.X := 0.430;
			MC_BR_MoveInPlane_Acp6D_0.Parameters.Position.Y := 0.420;
			MC_BR_MoveInPlane_Acp6D_0.Parameters.Path := 0;
			MC_BR_MoveInPlane_Acp6D_0.Parameters.Mode := 0;
			MC_BR_MoveInPlane_Acp6D_0.Execute := TRUE;
			IF MC_BR_MoveInPlane_Acp6D_0.Acknowledge THEN
				MC_BR_MoveInPlane_Acp6D_0.Execute := FALSE;
				em.substate := 10020;
			END_IF

		10020:
			em.description := 'Move Shuttle 4 towards workstation 2';
			MC_BR_MoveInPlane_Acp6D_0.Parameters.Acceleration := gAcp6DCtrl.Par.Acceleration;
			MC_BR_MoveInPlane_Acp6D_0.Parameters.Velocity := gAcp6DCtrl.Par.Velocity;
			MC_BR_MoveInPlane_Acp6D_0.Shuttle := ADR(gAcp6DCtrl.Status.ShuttleInfo[3].shuttleRef);
			MC_BR_MoveInPlane_Acp6D_0.Parameters.Position.X := 0.420;
			MC_BR_MoveInPlane_Acp6D_0.Parameters.Position.Y := 0.180;
			MC_BR_MoveInPlane_Acp6D_0.Parameters.Path := 0;
			MC_BR_MoveInPlane_Acp6D_0.Parameters.Mode := 0;
			MC_BR_MoveInPlane_Acp6D_0.Execute := TRUE;
			IF MC_BR_MoveInPlane_Acp6D_0.Acknowledge THEN
				MC_BR_MoveInPlane_Acp6D_0.Execute := FALSE;
				em.substate := 10025;
			END_IF

		10025:
			em.description := 'Move Shuttle 4 towards workstation 2';
			MC_BR_MoveInPlane_Acp6D_0.Parameters.Acceleration := gAcp6DCtrl.Par.Acceleration;
			MC_BR_MoveInPlane_Acp6D_0.Parameters.Velocity := gAcp6DCtrl.Par.Velocity;
			MC_BR_MoveInPlane_Acp6D_0.Shuttle := ADR(gAcp6DCtrl.Status.ShuttleInfo[3].shuttleRef);
			MC_BR_MoveInPlane_Acp6D_0.Parameters.Position.X := 0.430;
			MC_BR_MoveInPlane_Acp6D_0.Parameters.Position.Y := 0.180;
			MC_BR_MoveInPlane_Acp6D_0.Parameters.Path := 0;
			MC_BR_MoveInPlane_Acp6D_0.Parameters.Mode := 0;
			MC_BR_MoveInPlane_Acp6D_0.Execute := TRUE;
			IF MC_BR_MoveInPlane_Acp6D_0.Acknowledge THEN
				MC_BR_MoveInPlane_Acp6D_0.Execute := FALSE;
				em.substate := 10030;
			END_IF

		10030:
			em.description := 'Shuttle now move with the help of DanFossWork Task';
	END_CASE

END_ACTION

ACTION DanFossWork:
	// Setup

	CASE cm.state OF
		// Display station at image
		//'<foreignObject x="20" y="20" width="300" height="300"><img src="Media/statusGreen.png" height="300" width="300"/>'
		//brsstrcat(ADR(showWorkStations),ADR('<foreingObject x="'));
		//brdkStrCat(ADR(showWorkStations), ADR(testDraw));
		//brdkStrCat(ADR(showWorkStations),'<foreingObject x="');

		0:
			//Check what shuttle is on top of workstation
			FOR k := 0 TO NUM_SHUTTLES DO
				IF((gAcp6DCtrl.Status.ShuttleInfo[k].Position.X > pWorkStations.par.xLocation - MARGIN AND gAcp6DCtrl.Status.ShuttleInfo[k].Position.X < pWorkStations.par.xLocation + MARGIN) AND
					gAcp6DCtrl.Status.ShuttleInfo[k].Position.Y > pWorkStations.par.yLocation - MARGIN AND gAcp6DCtrl.Status.ShuttleInfo[k].Position.Y < pWorkStations.par.yLocation + MARGIN) THEN
					IF gAcp6DCtrl.Status.ShuttleInfo[k].State = mcACP6D_SH_STATE_IDLING THEN
						pWorkStations.par.tempShuttleID := k;
						IF pWorkStations.par.landBeforeProcess THEN
							cm.state := 10;
						ELSE
							cm.state := 20;
						END_IF
					END_IF
				END_IF
			END_FOR

		10:
			//Land shuttle if reguired
			pWorkStations.MC_BR_ShLevitation_Acp6D_0.Shuttle := ADR(gAcp6DCtrl.Status.ShuttleInfo[pWorkStations.par.tempShuttleID].shuttleRef);
			pWorkStations.MC_BR_ShLevitation_Acp6D_0.Parameters.Level := 0; //Land
			pWorkStations.MC_BR_ShLevitation_Acp6D_0.Parameters.Speed := REAL_TO_USINT(gAcp6DCtrl.Par.Velocity);
			pWorkStations.MC_BR_ShLevitation_Acp6D_0.Execute := TRUE;
			IF pWorkStations.MC_BR_ShLevitation_Acp6D_0.Done THEN
				pWorkStations.MC_BR_ShLevitation_Acp6D_0.Execute := FALSE;
				cm.state := 20;
			END_IF

		20:
			//Simulate process TON timer
			IF pWorkStations.status.oneshot THEN
				pWorkStations.TON_0.PT := REAL_TO_TIME(pWorkStations.par.processTime*1000/2);
			ELSE
				pWorkStations.TON_0.PT := REAL_TO_TIME(pWorkStations.par.processTime*1000);
			END_IF

			pWorkStations.TON_0.IN := TRUE;

			IF pWorkStations.TON_0.Q THEN
				pWorkStations.TON_0.IN := FALSE;
				pWorkStations.status.oneshot := FALSE;
				IF pWorkStations.par.landBeforeProcess THEN
					cm.state := 30;
				ELSE
					cm.state := 40;
				END_IF
			END_IF

		30:
			//Leviate shuttle if landed before process
			pWorkStations.MC_BR_ShLevitation_Acp6D_0.Shuttle := ADR(gAcp6DCtrl.Status.ShuttleInfo[pWorkStations.par.tempShuttleID].shuttleRef);
			pWorkStations.MC_BR_ShLevitation_Acp6D_0.Parameters.Level := 1; //Land
			pWorkStations.MC_BR_ShLevitation_Acp6D_0.Parameters.Speed := REAL_TO_USINT(gAcp6DCtrl.Par.Velocity);
			pWorkStations.MC_BR_ShLevitation_Acp6D_0.Execute := TRUE;
			IF pWorkStations.MC_BR_ShLevitation_Acp6D_0.Done THEN
				pWorkStations.MC_BR_ShLevitation_Acp6D_0.Execute := FALSE;
				cm.state := 20;
			END_IF

		40:
		//Move to fastLane X numbers of times and return
			IF pWorkStations.par.tempCounter >= pWorkStations.par.internalCounter THEN
				cm.state := 200;
			ELSE
				cm.state := 50;
			END_IF

		50:
			pWorkStations.MC_BR_MoveInPlane_Acp6D_0.Shuttle := ADR(gAcp6DCtrl.Status.ShuttleInfo[pWorkStations.par.tempShuttleID].shuttleRef);
			pWorkStations.MC_BR_MoveInPlane_Acp6D_0.Parameters.Velocity := gAcp6DCtrl.Par.Velocity;
			pWorkStations.MC_BR_MoveInPlane_Acp6D_0.Parameters.Acceleration := gAcp6DCtrl.Par.Acceleration;

			CASE i OF
				0:
					pWorkStations.MC_BR_MoveInPlane_Acp6D_0.Parameters.Position.X := 0.300;
					pWorkStations.MC_BR_MoveInPlane_Acp6D_0.Parameters.Position.Y := 0.180;
					IF pWorkStations.par.tempCounter > 0 THEN
						pWorkStations.MC_BR_MoveInPlane_Acp6D_0.Parameters.EndVelocity := gAcp6DCtrl.Par.Velocity;
					ELSE
						pWorkStations.MC_BR_MoveInPlane_Acp6D_0.Parameters.EndVelocity := 0;
					END_IF

				1:
					pWorkStations.MC_BR_MoveInPlane_Acp6D_0.Parameters.Position.X := 0.300;
					pWorkStations.MC_BR_MoveInPlane_Acp6D_0.Parameters.Position.Y := 0.420;
					IF pWorkStations.par.tempCounter > 0 THEN
						pWorkStations.MC_BR_MoveInPlane_Acp6D_0.Parameters.EndVelocity := 0;
					ELSE
						pWorkStations.MC_BR_MoveInPlane_Acp6D_0.Parameters.EndVelocity := gAcp6DCtrl.Par.Velocity;
					END_IF
			END_CASE

			pWorkStations.MC_BR_MoveInPlane_Acp6D_0.Parameters.Mode := 0; //Absolute
			pWorkStations.MC_BR_MoveInPlane_Acp6D_0.Parameters.Path := 0; //0 Diagonal, 1 First X then Y, 2 First Y then X
			pWorkStations.MC_BR_MoveInPlane_Acp6D_0.Execute := TRUE;
			IF pWorkStations.MC_BR_MoveInPlane_Acp6D_0.Acknowledge THEN
				pWorkStations.MC_BR_MoveInPlane_Acp6D_0.Execute := FALSE;
				IF i = 0 THEN
					cm.state := 55;
				ELSE
					cm.state := 60;
				END_IF
			END_IF

		55:
			pWorkStations.MC_BR_MoveInPlane_Acp6D_0.Shuttle := ADR(gAcp6DCtrl.Status.ShuttleInfo[pWorkStations.par.tempShuttleID].shuttleRef);
			pWorkStations.MC_BR_MoveInPlane_Acp6D_0.Parameters.Velocity := gAcp6DCtrl.Par.Velocity;
			pWorkStations.MC_BR_MoveInPlane_Acp6D_0.Parameters.Acceleration := gAcp6DCtrl.Par.Acceleration;
			pWorkStations.MC_BR_MoveInPlane_Acp6D_0.Parameters.EndVelocity := 0;

			pWorkStations.MC_BR_MoveInPlane_Acp6D_0.Parameters.Position.X := 0.300;
			pWorkStations.MC_BR_MoveInPlane_Acp6D_0.Parameters.Position.Y := 0.415;

			pWorkStations.MC_BR_MoveInPlane_Acp6D_0.Parameters.Mode := 0; //Absolute
			pWorkStations.MC_BR_MoveInPlane_Acp6D_0.Parameters.Path := 0; //0 Diagonal, 1 First X then Y, 2 First Y then X
			pWorkStations.MC_BR_MoveInPlane_Acp6D_0.Execute := TRUE;
			IF pWorkStations.MC_BR_MoveInPlane_Acp6D_0.Acknowledge THEN
				pWorkStations.MC_BR_MoveInPlane_Acp6D_0.Execute := FALSE;
				cm.state := 60;
			END_IF

		60:
			pWorkStations.MC_BR_MoveInPlane_Acp6D_0.Shuttle := ADR(gAcp6DCtrl.Status.ShuttleInfo[pWorkStations.par.tempShuttleID].shuttleRef);pWorkStations.par.tempShuttleID;
			pWorkStations.MC_BR_MoveInPlane_Acp6D_0.Parameters.Velocity := gAcp6DCtrl.Par.Velocity;
			pWorkStations.MC_BR_MoveInPlane_Acp6D_0.Parameters.Acceleration := gAcp6DCtrl.Par.Acceleration;
			pWorkStations.MC_BR_MoveInPlane_Acp6D_0.Parameters.EndVelocity := 0;

			pWorkStations.MC_BR_MoveInPlane_Acp6D_0.Parameters.Position.X := 0.060;
			pWorkStations.MC_BR_MoveInPlane_Acp6D_0.Parameters.Position.Y := 0.420;

			pWorkStations.MC_BR_MoveInPlane_Acp6D_0.Parameters.Mode := 0; //Absolute
			pWorkStations.MC_BR_MoveInPlane_Acp6D_0.Parameters.Path := 0; //0 Diagonal, 1 First X then Y, 2 First Y then X
			pWorkStations.MC_BR_MoveInPlane_Acp6D_0.Execute := TRUE;
			IF pWorkStations.MC_BR_MoveInPlane_Acp6D_0.Acknowledge THEN
				pWorkStations.MC_BR_MoveInPlane_Acp6D_0.Execute := FALSE;
				cm.state := 70;
			END_IF

		70:
			pWorkStations.MC_BR_MoveInPlane_Acp6D_0.Shuttle := ADR(gAcp6DCtrl.Status.ShuttleInfo[pWorkStations.par.tempShuttleID].shuttleRef);
			pWorkStations.MC_BR_MoveInPlane_Acp6D_0.Parameters.Velocity := gAcp6DCtrl.Par.Velocity;
			pWorkStations.MC_BR_MoveInPlane_Acp6D_0.Parameters.Acceleration := gAcp6DCtrl.Par.Acceleration;
			pWorkStations.MC_BR_MoveInPlane_Acp6D_0.Parameters.EndVelocity := 0;

			pWorkStations.MC_BR_MoveInPlane_Acp6D_0.Parameters.Position.X := 0.300;
			pWorkStations.MC_BR_MoveInPlane_Acp6D_0.Parameters.Position.Y := 0.060;

			pWorkStations.MC_BR_MoveInPlane_Acp6D_0.Parameters.Mode := 0; //Absolute
			pWorkStations.MC_BR_MoveInPlane_Acp6D_0.Parameters.Path := 2; //0 Diagonal, 1 First X then Y, 2 First Y then X
			pWorkStations.MC_BR_MoveInPlane_Acp6D_0.Execute := TRUE;
			IF pWorkStations.MC_BR_MoveInPlane_Acp6D_0.Acknowledge THEN
				pWorkStations.status.oneshot := FALSE;
				pWorkStations.MC_BR_MoveInPlane_Acp6D_0.Execute := FALSE;
				cm.state := 80;
			END_IF

		80:
			pWorkStations.MC_BR_MoveInPlane_Acp6D_0.Shuttle := ADR(gAcp6DCtrl.Status.ShuttleInfo[pWorkStations.par.tempShuttleID].shuttleRef);
			pWorkStations.MC_BR_MoveInPlane_Acp6D_0.Parameters.Velocity := gAcp6DCtrl.Par.Velocity;
			pWorkStations.MC_BR_MoveInPlane_Acp6D_0.Parameters.Acceleration := gAcp6DCtrl.Par.Acceleration;
			CASE i OF
				0:
					pWorkStations.MC_BR_MoveInPlane_Acp6D_0.Parameters.Position.X := 0.300;
					pWorkStations.MC_BR_MoveInPlane_Acp6D_0.Parameters.Position.Y := 0.060;
					IF pWorkStations.par.tempCounter+1 >= pWorkStations.par.internalCounter THEN
						pWorkStations.MC_BR_MoveInPlane_Acp6D_0.Parameters.EndVelocity := 0.5;
					ELSE
						pWorkStations.MC_BR_MoveInPlane_Acp6D_0.Parameters.EndVelocity := 0;
					END_IF

				1:
					pWorkStations.MC_BR_MoveInPlane_Acp6D_0.Parameters.Position.X := 0.300;
					pWorkStations.MC_BR_MoveInPlane_Acp6D_0.Parameters.Position.Y := 0.300;
					IF pWorkStations.par.tempCounter+1 >= pWorkStations.par.internalCounter THEN
						pWorkStations.MC_BR_MoveInPlane_Acp6D_0.Parameters.EndVelocity := 0;
					ELSE
						pWorkStations.MC_BR_MoveInPlane_Acp6D_0.Parameters.EndVelocity := 0.5;
					END_IF
			END_CASE

			pWorkStations.MC_BR_MoveInPlane_Acp6D_0.Parameters.Mode := 0; //Absolute
			pWorkStations.MC_BR_MoveInPlane_Acp6D_0.Parameters.Path := 0; //0 Diagonal, 1 First X then Y, 2 First Y then X

//			IF pWorkStations.par.tempCounter+1 >= pWorkStations.par.internalCounter THEN
//				pWorkStations.MC_BR_MoveInPlane_Acp6D_0.EndVelocity := 0;
//			ELSE
//				pWorkStations.MC_BR_MoveInPlane_Acp6D_0.EndVelocity := 0.5;
//			END_IF

			pWorkStations.MC_BR_MoveInPlane_Acp6D_0.Execute := TRUE;
			IF pWorkStations.MC_BR_MoveInPlane_Acp6D_0.Acknowledge THEN
				pWorkStations.status.oneshot := FALSE;
				pWorkStations.MC_BR_MoveInPlane_Acp6D_0.Execute := FALSE;
				pWorkStations.par.tempCounter := pWorkStations.par.tempCounter + 1;
				cm.state := 40;
			END_IF

		200:
			pWorkStations.MC_BR_MoveInPlane_Acp6D_0.Shuttle := ADR(gAcp6DCtrl.Status.ShuttleInfo[pWorkStations.par.tempShuttleID].shuttleRef);
			pWorkStations.MC_BR_MoveInPlane_Acp6D_0.Parameters.Velocity := gAcp6DCtrl.Par.Velocity;
			pWorkStations.MC_BR_MoveInPlane_Acp6D_0.Parameters.Acceleration := gAcp6DCtrl.Par.Acceleration;
			pWorkStations.MC_BR_MoveInPlane_Acp6D_0.Parameters.EndVelocity := 0;
			CASE i OF
				0:
					pWorkStations.MC_BR_MoveInPlane_Acp6D_0.Parameters.Position.X := 0.420;
					pWorkStations.MC_BR_MoveInPlane_Acp6D_0.Parameters.Position.Y := 0.060;

				1:
					pWorkStations.MC_BR_MoveInPlane_Acp6D_0.Parameters.Position.X := 0.420;
					pWorkStations.MC_BR_MoveInPlane_Acp6D_0.Parameters.Position.Y := 0.300;
			END_CASE

			pWorkStations.MC_BR_MoveInPlane_Acp6D_0.Parameters.Mode := 0; //Absolute
			pWorkStations.MC_BR_MoveInPlane_Acp6D_0.Parameters.Path := 1; //0 Diagonal, 1 First X then Y, 2 First Y then X
			//pWorkStations.MC_BR_MoveInPlane_Acp6D_0.EndVelocity := gAcp6DCtrl.Par.Velocity;
			pWorkStations.MC_BR_MoveInPlane_Acp6D_0.Execute := TRUE;
			IF pWorkStations.MC_BR_MoveInPlane_Acp6D_0.Acknowledge THEN
				pWorkStations.status.oneshot := FALSE;
				pWorkStations.MC_BR_MoveInPlane_Acp6D_0.Execute := FALSE;
				cm.state := 210;
			END_IF

		210:
			pWorkStations.MC_BR_MoveInPlane_Acp6D_0.Shuttle := ADR(gAcp6DCtrl.Status.ShuttleInfo[pWorkStations.par.tempShuttleID].shuttleRef);
			pWorkStations.MC_BR_MoveInPlane_Acp6D_0.Parameters.Velocity := gAcp6DCtrl.Par.Velocity;
			pWorkStations.MC_BR_MoveInPlane_Acp6D_0.Parameters.Acceleration := gAcp6DCtrl.Par.Acceleration;
			pWorkStations.MC_BR_MoveInPlane_Acp6D_0.Parameters.EndVelocity := 0;
			CASE i OF
				0:
					pWorkStations.MC_BR_MoveInPlane_Acp6D_0.Parameters.Position.X := 0.420;
					pWorkStations.MC_BR_MoveInPlane_Acp6D_0.Parameters.Position.Y := 0.180;

				1:
					pWorkStations.MC_BR_MoveInPlane_Acp6D_0.Parameters.Position.X := 0.420;
					pWorkStations.MC_BR_MoveInPlane_Acp6D_0.Parameters.Position.Y := 0.420;
			END_CASE

			pWorkStations.MC_BR_MoveInPlane_Acp6D_0.Parameters.Mode := 0; //Absolute
			pWorkStations.MC_BR_MoveInPlane_Acp6D_0.Parameters.Path := 1; //0 Diagonal, 1 First X then Y, 2 First Y then X
			pWorkStations.MC_BR_MoveInPlane_Acp6D_0.Parameters.EndVelocity := 0;
			pWorkStations.MC_BR_MoveInPlane_Acp6D_0.Execute := TRUE;
			IF pWorkStations.MC_BR_MoveInPlane_Acp6D_0.Acknowledge THEN
				pWorkStations.status.oneshot := FALSE;
				pWorkStations.MC_BR_MoveInPlane_Acp6D_0.Execute := FALSE;
				cm.state := 220;
			END_IF

		220:
			pWorkStations.MC_BR_MoveInPlane_Acp6D_0.Shuttle := ADR(gAcp6DCtrl.Status.ShuttleInfo[pWorkStations.par.tempShuttleID].shuttleRef);
			pWorkStations.MC_BR_MoveInPlane_Acp6D_0.Parameters.Velocity := gAcp6DCtrl.Par.Velocity;
			pWorkStations.MC_BR_MoveInPlane_Acp6D_0.Parameters.Acceleration := gAcp6DCtrl.Par.Acceleration;
			pWorkStations.MC_BR_MoveInPlane_Acp6D_0.Parameters.EndVelocity := 0;
			CASE i OF
				0:
					pWorkStations.MC_BR_MoveInPlane_Acp6D_0.Parameters.Position.X := 0.430;
					pWorkStations.MC_BR_MoveInPlane_Acp6D_0.Parameters.Position.Y := 0.180;

				1:
					pWorkStations.MC_BR_MoveInPlane_Acp6D_0.Parameters.Position.X := 0.430;
					pWorkStations.MC_BR_MoveInPlane_Acp6D_0.Parameters.Position.Y := 0.420;
			END_CASE

			pWorkStations.MC_BR_MoveInPlane_Acp6D_0.Parameters.Mode := 0; //Absolute
			pWorkStations.MC_BR_MoveInPlane_Acp6D_0.Parameters.Path := 1; //0 Diagonal, 1 First X then Y, 2 First Y then X
			//pWorkStations.MC_BR_MoveInPlane_Acp6D_0.EndVelocity := gAcp6DCtrl.Par.Velocity;
			pWorkStations.MC_BR_MoveInPlane_Acp6D_0.Execute := TRUE;
			IF pWorkStations.MC_BR_MoveInPlane_Acp6D_0.Acknowledge THEN
				pWorkStations.status.oneshot := FALSE;
				pWorkStations.MC_BR_MoveInPlane_Acp6D_0.Execute := FALSE;
				pWorkStations.par.tempCounter := 0;
				cm.state := 0;
			END_IF

	END_CASE

	//Calls
	pWorkStations.MC_BR_MoveInPlane_Acp6D_0();
	pWorkStations.MC_BR_ShLevitation_Acp6D_0();
	pWorkStations.TON_0();
	cm();

END_ACTION
```
